(* CODESYS project CtaAppModBus_1.0.0.0.library
   Description: Modbus Library der CTA
   Version: 1.0.0.0
   Title: CtaAppModbus
   Author: SIS
   Company: CTA
   Placeholder: CtaAppModbus
   DocFormat: reStructuredText
   CompiledLibraryCompatibilityVersion: CODESYS V3.5 SP16 Patch 3
   LanguageModelAttribute: qualified-access-only
   DefaultNamespace: CtaAppModbus

Project tree, tasks and I/O mapping:
  libraries: Standard, 3.5.18.0 (System); CtaVisSymbols, 1.0.0.0 (CTA); CtaSysConfig, 1.0.0.0 (CTA); CtaAppTime, 1.0.0.0 (CTA); CtaAppBmk, 1.0.0.0 (CTA); VisuSymbols, 4.5.0.0 (System); VisuDialogs, * (System); ModbusFB, 4.3.0.0 (3S - Smart Software Solutions GmbH); IoDrvEthernet, 4.2.0.0 (3S - Smart Software Solutions GmbH); CtaVisHelp, 1.0.0.0 (CTA)
  40 Visualizations/
    HELPER/
      visualisation VIS_IP_INPUT
      visualisation VIS_IP_PARAMETER
      visualisation VIS_IP_PARAMETER_QUERRY
      visualisation VIS_IP_PARAMETER_BASE
    CLIENTMANAGER/
      LINE/
        visualisation VIS_CLIENT_LINE_QUERRY
        visualisation VIS_CLIENT_LINE
      OVERWIEV/
        visualisation VIS_CLIENT_MANAGER_OVERWIEV_QUERRY
        visualisation VIS_CLIENT_MANAGER_TABLE
        visualisation VIS_CLIENT_MANAGER_OVERWIEV
      MENÜ/
        visualisation VIS_CLIENTMANAGER_MENÜ
      visualisation DIA_CLIENT_MANAGER
      PARAMETER/
        visualisation VIS_CLIENT_MANAGER_PARAMETER
      TCP/
        PARAMETER/
          visualisation VIS_CLIENT_MANAGER_PARAMETER_TCP
          visualisation VIS_CLIENT_MANAGER_PARAMETER_TCP_QUERY
      RTU/
        PARAMETER/
          visualisation VIS_CLIENT_MANAGER_PARAMETER_RTU
          visualisation VIS_CLIENT_MANAGER_PARAMETER_RTU_QUERY
          TEXTLIST/
            text list TEXT_DTR_CONTROL
            text list TEXT_RTS_CONTROL
            text list TEXT_STOPBITS
            text list TXT_COMPORT
    MBJOB/
      visualisation VIS_JOB_QUERRY
      visualisation VIS_JOB
    CLIENT/
      TCP/
        PARAMETER/
          visualisation VIS_CLIENT_PARAMETER_TCP
          visualisation VIS_CLIENT_PARAMETER_TCP_QUERY
          visualisation VIS_CLIENT_PARAMETER_TCP_TEMP
      RTU/
        PARAMETER/
          visualisation VIS_CLIENT_PARAMETER_RTU
          visualisation VIS_CLIENT_PARAMETER_RTU_QUERY
          visualisation VIS_CLIENT_PARAMETER_RTU_TEMP
      CLIENT/
        visualisation DIA_CLIENT
        MENÜ/
          visualisation VIS_CLIENT_MENÜ
        OVERWIEV/
          visualisation VIS_CLIENT_OVERWIEV
          visualisation VIS_CLIENT_OVERWIEV_QUERY
        PARAMETER/
          visualisation VIS_CLIENT_PARAMETER
        JOBS/
          visualisation VIS_CLIENT_JOBS_TABLE
          visualisation VIS_CLIENT_JOBS_QUERRY
          visualisation VIS_CLIENT_JOBS
    SERVER/
      visualisation DIA_SERVER
  30 Program Organization Units/
    CLIENT/
      TCP/
        function block FB_MB_CLIENT_TCP [ST]: NODE_ID, ENABLE, TIMEOUT, READ_DELAY, WRITE_DELAY, IP_ADRESS, actConfig, PORT, P_fbtWriteDelay, P_fbuiPort, P_fbtTimeOut, P_fbusiNodeId, P_fbxEnable, P_fbstIpAdress, P_fbtReadDelay
      RTU/
        function block FB_MB_CLIENT_RTU [ST]: TIMEOUT, NODE_ID, READ_DELAY, WRITE_DELAY, actConfig, ENABLE, P_fbtReadDelay, P_fbtTimeOut, P_fbtWriteDelay, P_fbusiNodeId, P_fbxEnable
      BASE/
        function block FB_MB_CLIENT [ST]: ADD_MODBUS_JOB, CHECK_IF_JOB_EXIST, CREATE_JOB, GET_NEXT_JOB, DESTROY_JOB, AllJobsDone, GET_READY, BIG_SYBIL, LOW_SYBIL, SELF, CALL_AFTER_LAST_JOB_DONE, BASE_MBJOB, COUNT, ERROR, ERROR_ID, EXEPTION_CODE, AY_ITF_MBJOB_VIS, ExecuteTime, RELOAD_ARRAY, IsCurrentCall, CONFIRM_ALL_JOBS_DONE
    MBJOB/
      function block FB_MBJOB [ST]: byMbFunction, PARENT, BIG_SYBIL, pByte, wQuantity, DESTROY, wMbAdress, LOW_SYBIL, SELF
    FC/
      function FcBytePointToWordValue [ST]
      function FcBytePointToBoolValue [ST]
      function fcStringIPtoByteArray [ST]
      function fcSetInitialIPString [ST]
      function fcCheckIp [ST]
    CLIENTMANAGER/
      RTU/
        function block FB_MB_CLIENTMANAGER_RTU [ST]: actConfig, actGetError, P_fbenRTSControl, actCallFunctions, actCheckBusy, actDelays, actExecuteFunction, P_fbenStopBits, P_fbxRtuAscii, P_fbbyDataBits, P_fbdwBaudrate, P_fbenDTRControl, P_fbenParity, P_fbenPort
      TCP/
        function block FB_MB_CLIENTMANAGER_TCP [ST]: actGetError, actCheckBusy, actExecuteFunction, actDelays, actCallFunctions
      BASE/
        function block FB_MB_CLIENTMANAGER [ST]: ITF_BASE_CLIENT, ADD_MODBUS_CLIENT, CHECK_IF_EXIST, RELOAD_ARRAY, AY_ITF_MBCLIENT_VIS, OperationTime
    SERVER/
      function block fbModBusServer [ST]: actConfig, actModBusServerTcp, actModBusServerUdp, actModBusServerSerial, metGetCoil, metSetDiscretInput, metGetHoldingRegister, metSetInputRegister, metAddSerialControll, metAddTcpControll, metAddUdpControll, metSetHoldingRegister, metSetCoil
      function block FB_SERVER [ST]: actConfig, metGetCoil, metGetHoldingRegister, metSetCoil, metSetDiscretInput, metSetHoldingRegister, metSetInputRegister, actDataModel, P_Serial_fbbyDataBits, P_Serial_fbdwBaudrate, P_Serial_fbenDTRControl, P_Serial_fbenParity, P_Serial_fbenRTSControl, P_Serial_fbenStopBits, P_Serial_fbusiNodeId, P_Serial_fbxEnable, P_Serial_fbxRtuAscii, P_Serial_fbxEnableWatchDog, P_Serial_fbtWatchDog, P_Serial_fbenPort, P_Tcp_fbxEnable, P_Tcp_fbwPort, P_Tcp_fbxEnableWatchDog, P_Tcp_fbtWatchDog, P_Tcp_fbstInterface
  00000000-0000-0000-0000-000000000000|D:\CoDeSys\LibrariesV3\trunk\Intern\CAA\CAA Template\3.4.0.0 draft\Placeholder.xml
  00000000-0000-0000-0000-000000000000|D:\CoDeSys\LibrariesV3\trunk\Intern\CAA\CAA Template\3.2.0.3 draft\Prefix.pdf
  00000000-0000-0000-0000-000000000000|D:\CoDeSys\LibrariesV3\trunk\Intern\CAA\CAA Template\3.5.2.0 draft\Placeholder.xml
  20 Structs/
    SERVER/
      PARAMETER/
        data type scModBusServerParameter
        TCP/
          data type scTcp
        SERIAL/
          data type scSerial
    CLIENT/
      NETWORK/
        data type scTcpClientParameter
      SERIAL/
        data type scSerialPortParameter
        data type scSerialClientParameter
  50 Images/
  10 Documenation/
    global variables VersionHistory
    global variables readMe
  21 Interface/
    CLIENTMANAGER/
      RTU/
        interface ITF_MB_CLIENTMANAGER_RTU: P_fbenStopBits, P_fbenPort, P_fbdwBaudrate, P_fbbyDataBits, P_fbenParity, P_fbenDTRControl, P_fbenRTSControl, P_fbxRtuAscii
      BASE/
        interface ITF_MB_CLIENTMANAGER: OperationTime, ITF_BASE_CLIENT, AY_ITF_MBCLIENT_VIS, RELOAD_ARRAY
      TCP/
        interface ITF_MB_CLIENTMANAGER_TCP
    MBJOB/
      interface ITF_MBJOB: PARENT, DESTROY, BIG_SYBIL, LOW_SYBIL, SELF, byMbFunction, pByte, wMbAdress, wQuantity
    CLIENT/
      BASE/
        interface ITF_CLIENT: CHECK_IF_JOB_EXIST, CREATE_JOB, DESTROY_JOB, GET_NEXT_JOB, GET_READY, AllJobsDone, BIG_SYBIL, LOW_SYBIL, SELF, BASE_MBJOB, COUNT, ADD_MODBUS_JOB, ERROR, ERROR_ID, EXEPTION_CODE, AY_ITF_MBJOB_VIS, ExecuteTime, RELOAD_ARRAY, IsCurrentCall, CONFIRM_ALL_JOBS_DONE, CALL_AFTER_LAST_JOB_DONE
      RTU/
        interface ITF_MB_CLIENT_RTU: ENABLE, P_fbxEnable, P_fbusiNodeId, P_fbtTimeOut, P_fbtReadDelay, P_fbtWriteDelay, NODE_ID, TIMEOUT, READ_DELAY, WRITE_DELAY
      TCP/
        interface ITF_MB_CLIENT_TCP: ENABLE, NODE_ID, TIMEOUT, READ_DELAY, WRITE_DELAY, IP_ADRESS, PORT, P_fbxEnable, P_fbusiNodeId, P_fbtTimeOut, P_fbtReadDelay, P_fbtWriteDelay, P_fbuiPort, P_fbstIpAdress
    SERVER/
      interface ITF_SERVER: metGetCoil, metGetHoldingRegister, metSetCoil, metSetDiscretInput, metSetHoldingRegister, metSetInputRegister
      interface ITF_SERVER_PARA: P_Serial_fbxEnable, P_Serial_fbusiNodeId, P_Serial_fbdwBaudrate, P_Serial_fbbyDataBits, P_Serial_fbenParity, P_Serial_fbenStopBits, P_Serial_fbenDTRControl, P_Serial_fbenRTSControl, P_Serial_fbxRtuAscii, P_Serial_fbxEnableWatchDog, P_Serial_fbtWatchDog, P_Serial_fbenPort, P_Tcp_fbxEnable, P_Tcp_fbwPort, P_Tcp_fbxEnableWatchDog, P_Tcp_fbtWatchDog, P_Tcp_fbstInterface
  11 Library Parameter/
  12 Konstanten/
  60 Textlisten/
    SERIAL/
      text list txtPhysikalLayer
      text list txtParity
      text list txtHandshake
      text list txtStopBits
  13 Globale Variablen/
  text list GlobalTextList
*)

// 20 Structs/SERVER/PARAMETER/scModBusServerParameter
TYPE scModBusServerParameter :
    STRUCT
        scSerial    :   scSerial;
        scTcp       :   scTcp;
    END_STRUCT
END_TYPE

// 20 Structs/SERVER/PARAMETER/TCP/scTcp
TYPE scTcp :
    STRUCT
        fbxEnable           :   CtaSysConfig.fbBOOL;           // Tcp Server Enable    
        fbwPort             :   CtaSysConfig.fbWORD;           // Tcp Server Port
        fbxEnableWatchDog   :   CtaSysConfig.fbBOOL;           // WatchDog Enable
        fbtWatchDog         :   CtaSysConfig.fbTIME;           // WatchDog Time
		fbstInterface		:	CtaSysConfig.fbSTRING40;	   // Interface Name
    END_STRUCT
END_TYPE

// 20 Structs/SERVER/PARAMETER/SERIAL/scSerial
TYPE scSerial :
    STRUCT
        fbxEnable           				:   CtaSysConfig.fbBOOL;        // Serial Server Enable
        fbxEnableWatchDog   				:   CtaSysConfig.fbBOOL;        // WatchDog Enable
        fbtWatchDog         				:   CtaSysConfig.fbTIME;        // WatchDog Time		
		fbenPort							:	CtaSysConfig.fbINT;			// PORT NONE , COM1, COM2 ...
		fbusiNodeId							:	CtaSysConfig.fbUSINT;      	// Serial Server Id  
		fbdwBaudrate						:	CtaSysConfig.fbDWORD;		// Baudrate 
		fbbyDataBits						:	CtaSysConfig.fbBYTE;		// Data Bits
		fbenParity							:	CtaSysConfig.fbBYTE;		// Parity
		fbenStopBits						:	CtaSysConfig.fbBYTE;		// Stopbits
		fbenDTRControl						:	CtaSysConfig.fbBYTE;		// DTR Control
		fbenRTSControl						:	CtaSysConfig.fbBYTE;		// RTS Control
		fbxRtuAscii							:	CtaSysConfig.fbBOOL;		// RTU = FALSE , ASCII = TRUE
    END_STRUCT
END_TYPE

// 20 Structs/CLIENT/NETWORK/scTcpClientParameter
TYPE scTcpClientParameter :
    STRUCT
        fbxEnable					:	CtaSysConfig.fbBOOL;        // Serial Server Enable       
        fbusiNodeId					:	CtaSysConfig.fbUSINT;     	// Serial Server Id  
        fbtTimeOut					:	CtaSysConfig.fbTIME;        // Timeout Time
        fbtReadDelay				:	CtaSysConfig.fbTIME;      	// Read Delay        
        fbtWriteDelay				:	CtaSysConfig.fbTIME;     	// Write Delay 	
		fbuiPort					:	CtaSysConfig.fbUINT;      	// Port Nr  
		fbstIpAdress				:	CtaSysConfig.fbSTRING40;    // IP Adresse   
    END_STRUCT
END_TYPE

// 20 Structs/CLIENT/SERIAL/scSerialPortParameter
TYPE scSerialPortParameter :
    STRUCT 
		fbenPort							:	CtaSysConfig.fbINT;			// PORT NONE , COM1, COM2 ...
		fbdwBaudrate						:	CtaSysConfig.fbDWORD;		// Baudrate 
		fbbyDataBits						:	CtaSysConfig.fbBYTE;		// Data Bits
		fbenParity							:	CtaSysConfig.fbBYTE;		// Parity
		fbenStopBits						:	CtaSysConfig.fbBYTE;		// Stopbits
		fbenDTRControl						:	CtaSysConfig.fbBYTE;		// DTR Control
		fbenRTSControl						:	CtaSysConfig.fbBYTE;		// RTS Control
		fbxRtuAscii							:	CtaSysConfig.fbBOOL;		// RTU = FALSE , ASCII = TRUE
    END_STRUCT
END_TYPE

// 20 Structs/CLIENT/SERIAL/scSerialClientParameter
TYPE scSerialClientParameter :
    STRUCT
        fbxEnable					:	CtaSysConfig.fbBOOL;       // Serial Server Enable        
        fbusiNodeId					:	CtaSysConfig.fbUSINT;      // Serial Server Id        
        fbtTimeOut					:	CtaSysConfig.fbTIME;       // Timeout Time
		fbtReadDelay				:	CtaSysConfig.fbTIME; 	   // Read Delay
		fbtWriteDelay				:	CtaSysConfig.fbTIME;	   // Write Delay
    END_STRUCT
END_TYPE

// 10 Documenation/VersionHistory
(* 

.. image:: ../../Images/CTA_Logo.jpg
   :align: right
   :width: 15% 

**Vorlage**   


============ =========== =========== ============================================
**Date**     **Version** **Author**  **Change**
------------ ----------- ----------- --------------------------------------------
04.03.2021   0.0.0.0     SIS         Vorlage erstellt

============ =========== =========== ============================================


*)
VAR_GLOBAL
    stInfo : STRING:= '0.0.0.0, Vorlage, CTA';
END_VAR

// 10 Documenation/readMe
(*

**ReadMe**
 
|	**Empfehlung**
|
|	Dokumentrieren Sie die Library für eine nachhaltige Entwicklung
|     
| *Beispiel* 
|
| Dies ist die Vorlage Library der CTA. Erstellen Sie ihre Library anhand dieser Vorlage.
*)

VAR_GLOBAL
    xReadMeDone              :   BOOL;
END_VAR

// 30 Program Organization Units/MBJOB/FB_MBJOB
{attribute 'enable_dynamic_creation'}
FUNCTION_BLOCK FB_MBJOB IMPLEMENTS ITF_MBJOB
VAR_OUTPUT
END_VAR
VAR
	_xConfirmExecute:	BOOL;
	_byMbFunction	:	BYTE;
	_wMbAdress		:	WORD;
	_pByte			:	POINTER TO BYTE;
	_wQuantity		:	WORD;	
	_ITF_BIG_SYBIL	:	ITF_MBJOB;
	_ITF_LOW_SYBIL	:	ITF_MBJOB;
	_ITF_PARENT		:	ITF_CLIENT;
END_VAR

PROPERTY byMbFunction : BYTE
GET
byMbFunction := _byMbFunction;
END_GET
SET
_byMbFunction := byMbFunction;
END_SET
END_PROPERTY

PROPERTY PARENT : ITF_CLIENT
SET
_ITF_PARENT := PARENT;
END_SET
END_PROPERTY

{attribute 'estimated-stack-usage' := '104'}
PROPERTY BIG_SYBIL : ITF_MBJOB
GET
BIG_SYBIL := _ITF_BIG_SYBIL;
END_GET
SET
_ITF_BIG_SYBIL := BIG_SYBIL;
IF __QUERYINTERFACE(_ITF_BIG_SYBIL,_ITF_BIG_SYBIL) THEN
	IF _ITF_BIG_SYBIL.LOW_SYBIL <> SELF THEN
		_ITF_BIG_SYBIL.LOW_SYBIL := THIS^;
	END_IF;
END_IF;
END_SET
END_PROPERTY

PROPERTY pByte : POINTER TO BYTE
GET
pByte := _pByte;
END_GET
SET
_pByte := pByte;
END_SET
END_PROPERTY

PROPERTY wQuantity : WORD
GET
wQuantity := _wQuantity;
END_GET
SET
_wQuantity := wQuantity;
END_SET
END_PROPERTY

METHOD DESTROY
VAR
	pSelf	:	POINTER TO FB_MBJOB;
END_VAR
IF __QUERYINTERFACE(_ITF_BIG_SYBIL,_ITF_BIG_SYBIL) THEN
	_ITF_BIG_SYBIL.LOW_SYBIL := _ITF_LOW_SYBIL;
END_IF;

IF __QUERYINTERFACE(_ITF_LOW_SYBIL,_ITF_LOW_SYBIL) THEN
	_ITF_LOW_SYBIL.BIG_SYBIL := _ITF_BIG_SYBIL;
END_IF;

IF __QUERYINTERFACE(_ITF_PARENT,_ITF_PARENT) THEN
	_ITF_PARENT.RELOAD_ARRAY(TRUE,FALSE,FALSE);
END_IF;

pSelf := THIS;

__DELETE(pSelf);
END_METHOD

PROPERTY wMbAdress : WORD
SET
_wMbAdress := wMbAdress;
END_SET
GET
wMbAdress := _wMbAdress;
END_GET
END_PROPERTY

{attribute 'estimated-stack-usage' := '104'}
PROPERTY LOW_SYBIL : ITF_MBJOB
GET
LOW_SYBIL := _ITF_LOW_SYBIL;
END_GET
SET
_ITF_LOW_SYBIL := LOW_SYBIL;
IF __QUERYINTERFACE(_ITF_LOW_SYBIL,_ITF_LOW_SYBIL) THEN
	IF _ITF_LOW_SYBIL.BIG_SYBIL <> SELF THEN
		_ITF_LOW_SYBIL.BIG_SYBIL := THIS^;
	END_IF;
END_IF;
END_SET
END_PROPERTY

PROPERTY SELF : ITF_MBJOB
GET
SELF := THIS^;
END_GET
END_PROPERTY

END_FUNCTION_BLOCK

// 21 Interface/MBJOB/ITF_MBJOB
INTERFACE ITF_MBJOB EXTENDS __System.IQUERYINTERFACE

PROPERTY PARENT : ITF_CLIENT
SET
END_SET
END_PROPERTY

METHOD DESTROY
END_METHOD

PROPERTY BIG_SYBIL : ITF_MBJOB
GET
END_GET
SET
END_SET
END_PROPERTY

PROPERTY LOW_SYBIL : ITF_MBJOB
GET
END_GET
SET
END_SET
END_PROPERTY

PROPERTY SELF : ITF_MBJOB
GET
END_GET
END_PROPERTY

PROPERTY byMbFunction : BYTE
SET
END_SET
GET
END_GET
END_PROPERTY

PROPERTY pByte : POINTER TO BYTE
SET
END_SET
GET
END_GET
END_PROPERTY

PROPERTY wMbAdress : WORD
SET
END_SET
GET
END_GET
END_PROPERTY

PROPERTY wQuantity : WORD
GET
END_GET
SET
END_SET
END_PROPERTY

END_INTERFACE

// 21 Interface/CLIENT/BASE/ITF_CLIENT
INTERFACE ITF_CLIENT  EXTENDS CtaAppBmk.ITF_BMK

METHOD CHECK_IF_JOB_EXIST : BOOL
VAR_INPUT
	_byMbFunction	:	BYTE;
	_wMbAdress		:	WORD;
	_pByte			:	POINTER TO BYTE;
	_wQuantity		:	WORD;	
END_VAR
END_METHOD

METHOD CREATE_JOB : BOOL
VAR_INPUT
	_byMbFunction	:	BYTE;
	_wMbAdress		:	WORD;
	_pData			:	POINTER TO BYTE;
	_wQuantity		:	WORD;		
END_VAR
END_METHOD

METHOD DESTROY_JOB : BOOL
VAR_INPUT
	_byMbFunction	:	BYTE;
	_wMbAdress		:	WORD;
	_pData			:	POINTER TO BYTE;
	_wQuantity		:	WORD;		
END_VAR
END_METHOD

METHOD GET_NEXT_JOB : BOOL
VAR_OUTPUT
	_byMbFunction	:	BYTE;
	_wMbAdress		:	WORD;
	_pByte			:	POINTER TO BYTE;
	_wQuantity		:	WORD;	
END_VAR
END_METHOD

METHOD GET_READY : BOOL
VAR_INPUT
END_VAR
END_METHOD

PROPERTY AllJobsDone : BOOL
GET
END_GET
END_PROPERTY

PROPERTY BIG_SYBIL : ITF_CLIENT
GET
END_GET
SET
END_SET
END_PROPERTY

PROPERTY LOW_SYBIL : ITF_CLIENT
GET
END_GET
SET
END_SET
END_PROPERTY

PROPERTY SELF : ITF_CLIENT
GET
END_GET
END_PROPERTY

PROPERTY BASE_MBJOB : ITF_MBJOB
GET
END_GET
END_PROPERTY

PROPERTY COUNT : UINT
GET
END_GET
END_PROPERTY

METHOD ADD_MODBUS_JOB
VAR_INPUT
	ITF_MBJOB_IN	:	ITF_MBJOB;
END_VAR
END_METHOD

PROPERTY ERROR : BOOL
SET
END_SET
GET
END_GET
END_PROPERTY

PROPERTY ERROR_ID : ModbusFB.Error
SET
END_SET
GET
END_GET
END_PROPERTY

PROPERTY EXEPTION_CODE : ModbusFB.ExceptionCodes
SET
END_SET
GET
END_GET
END_PROPERTY

PROPERTY AY_ITF_MBJOB_VIS : ARRAY[0..9] OF ITF_MBJOB
GET
END_GET
END_PROPERTY

PROPERTY ExecuteTime : LTIME
GET
END_GET
END_PROPERTY

METHOD RELOAD_ARRAY
VAR_INPUT
	xInit				:	BOOL;
	xLoadNext10			:	BOOL;
	xLoadLast10			:	BOOL;
END_VAR
END_METHOD

PROPERTY IsCurrentCall : BOOL
GET
END_GET
END_PROPERTY

PROPERTY CONFIRM_ALL_JOBS_DONE : BOOL
GET
END_GET
END_PROPERTY

METHOD CALL_AFTER_LAST_JOB_DONE
VAR_INPUT
END_VAR
END_METHOD

END_INTERFACE

// 30 Program Organization Units/CLIENT/TCP/FB_MB_CLIENT_TCP
FUNCTION_BLOCK FB_MB_CLIENT_TCP EXTENDS FB_MB_CLIENT IMPLEMENTS ITF_MB_CLIENT_TCP
VAR_OUTPUT
END_VAR
VAR
	(* Config *)
	fbConfigFile				:	CtaSysConfig.fbConfigFile;
	scParameter                	: 	scTcpClientParameter;
END_VAR

(* Config File *)
actConfig();

PROPERTY NODE_ID : USINT
GET
NODE_ID := scParameter.fbusiNodeId.proValue;
END_GET
END_PROPERTY

PROPERTY ENABLE : BOOL
GET
ENABLE := scParameter.fbxEnable.proValue;
END_GET
END_PROPERTY

PROPERTY TIMEOUT : TIME
GET
TIMEOUT := scParameter.fbtTimeOut.proValue;
END_GET
END_PROPERTY

PROPERTY READ_DELAY : TIME
GET
READ_DELAY := scParameter.fbtReadDelay.proValue;
END_GET
END_PROPERTY

PROPERTY WRITE_DELAY : TIME
GET
WRITE_DELAY := scParameter.fbtWriteDelay.proValue;
END_GET
END_PROPERTY

PROPERTY IP_ADRESS : STRING(15)
GET
IP_ADRESS := scParameter.fbstIpAdress.proValue;
END_GET
END_PROPERTY

ACTION actConfig:
(* Config File *)
fbConfigFile();

scParameter.fbxEnable		(_usiParaNr := 1,itfConfigFb := fbConfigFile										);		
scParameter.fbusiNodeId		(_usiParaNr := 2,itfConfigFb := fbConfigFile,_MinInit := 0	  , _MaxInit := 255		);		
scParameter.fbtTimeOut		(_usiParaNr := 3,itfConfigFb := fbConfigFile,_MinInit := T#0MS, _MaxInit := T#5M 	);		
scParameter.fbtReadDelay	(_usiParaNr := 4,itfConfigFb := fbConfigFile,_MinInit := T#0MS, _MaxInit := T#5M 	);		
scParameter.fbtWriteDelay	(_usiParaNr := 5,itfConfigFb := fbConfigFile,_MinInit := T#0MS, _MaxInit := T#5M 	);	
scParameter.fbuiPort		(_usiParaNr := 6,itfConfigFb := fbConfigFile										);
scParameter.fbstIpAdress	(_usiParaNr := 7,itfConfigFb := fbConfigFile										);

(* Check Ip *)
IF scParameter.fbstIpAdress.proStateChanged THEN
	IF NOT fcCheckIp(scParameter.fbstIPAdress.proValue) THEN
		fcSetInitialIPString(scParameter.fbstIpAdress);
	END_IF;
END_IF;
END_ACTION

PROPERTY PORT : UINT
GET
PORT := scParameter.fbuiPort.proValue;
END_GET
END_PROPERTY

PROPERTY P_fbtWriteDelay : CtaSysConfig.ITF_DATATYPE
GET
P_fbtWriteDelay := scParameter.fbtWriteDelay;
END_GET
END_PROPERTY

PROPERTY P_fbuiPort : CtaSysConfig.ITF_DATATYPE
GET
P_fbuiPort := scParameter.fbuiPort;
END_GET
END_PROPERTY

PROPERTY P_fbtTimeOut : CtaSysConfig.ITF_DATATYPE
GET
P_fbtTimeOut := scParameter.fbtTimeOut;
END_GET
END_PROPERTY

PROPERTY P_fbusiNodeId : CtaSysConfig.ITF_DATATYPE
GET
P_fbusiNodeId := scParameter.fbusiNodeId;
END_GET
END_PROPERTY

PROPERTY P_fbxEnable : CtaSysConfig.ITF_DATATYPE
GET
P_fbxEnable := scParameter.fbxEnable;
END_GET
END_PROPERTY

PROPERTY P_fbstIpAdress : CtaSysConfig.ITF_DATATYPE
GET
P_fbstIpAdress := scParameter.fbstIpAdress;
END_GET
END_PROPERTY

PROPERTY P_fbtReadDelay : CtaSysConfig.ITF_DATATYPE
GET
P_fbtReadDelay := scParameter.fbtReadDelay;
END_GET
END_PROPERTY

END_FUNCTION_BLOCK

// 30 Program Organization Units/CLIENT/BASE/FB_MB_CLIENT
FUNCTION_BLOCK FB_MB_CLIENT EXTENDS CtaAppBmk.fbBMK IMPLEMENTS ITF_CLIENT
VAR_OUTPUT
	udiDynMem					:	UDINT;
	xAllJobsDone				:	BOOL;
	xConfirmAllJobsDone			:	BOOL;
END_VAR             			
VAR                 			
	_ITF_BIG_SYBIL				:	ITF_CLIENT;
	_ITF_LOW_SYBIL				:	ITF_CLIENT;
	                			
	_BASE_MBU_JOB				:	ITF_MBJOB;
	_TEMP_REG_JOB				:	ITF_MBJOB;
	_TEMP_MBU_JOB				:	ITF_MBJOB;	
	
	_COUNT						:	UINT;
	_udiDynMemTemp				:	UDINT;
	xGetReadyCalled				:	BOOL;
	xNoChangeHappen				:	BOOL;
	
	xErrorHappen				:	BOOL;
	eErrorID					:	ModbusFB.Error;
	eExeptionCode				:	ModbusFB.ExceptionCodes;
	
	fbTimeStop					:	CtaAppTime.fbTimeMeasurement;
	ltTime						:	LTIME;
	
	_ayITF_MBJOB_VIS			:	ARRAY[0..9] OF ITF_MBJOB;
END_VAR

METHOD ADD_MODBUS_JOB
VAR_INPUT
	ITF_MBJOB_IN	:	ITF_MBJOB;
END_VAR
VAR
	ITF_TEMP		:	ITF_MBJOB;
	ITF_TEMP_BIG	:	ITF_MBJOB;
	ITF_TEMP_LOW	:	ITF_MBJOB;
	xDone			:	BOOL;
END_VAR
(* Check if Valid Interface Input *)
IF __QUERYINTERFACE(ITF_MBJOB_IN,ITF_MBJOB_IN) THEN
	ITF_MBJOB_IN.PARENT := THIS^;
	(* Check if Valid Interface Base*)
	IF __QUERYINTERFACE(_BASE_MBU_JOB,_BASE_MBU_JOB) THEN
		(* Check if Valid Interface Temporary registration *)
		IF __QUERYINTERFACE(_TEMP_REG_JOB,ITF_TEMP) THEN
			REPEAT
				(* Get Big Sybil of registration *)
				IF __QUERYINTERFACE(ITF_TEMP.BIG_SYBIL,ITF_TEMP_BIG) THEN
					(* Check if Function Code is Lower or Bigger *)
					IF ITF_MBJOB_IN.byMbFunction <= ITF_TEMP.byMbFunction AND
						ITF_MBJOB_IN.byMbFunction >= ITF_TEMP_BIG.byMbFunction THEN
						(* Check if Adress is Lower *)
						IF ITF_MBJOB_IN.wMbAdress <= ITF_TEMP.wMbAdress THEN
							(* Check if Adress is Bigger and update if yes*)
							IF ITF_MBJOB_IN.wMbAdress >= ITF_TEMP_BIG.wMbAdress THEN
								ITF_MBJOB_IN.BIG_SYBIL := ITF_TEMP.BIG_SYBIL;
								ITF_MBJOB_IN.LOW_SYBIL := ITF_TEMP;
								xDone	 := TRUE;							
							END_IF;
						(* Adress is Bigger update *)
						ELSE
							IF __QUERYINTERFACE(ITF_TEMP.LOW_SYBIL,ITF_TEMP_LOW) THEN
								IF ITF_MBJOB_IN.byMbFunction < ITF_TEMP_LOW.byMbFunction OR
									(ITF_MBJOB_IN.byMbFunction = ITF_TEMP_LOW.byMbFunction AND
									ITF_MBJOB_IN.wMbAdress <= ITF_TEMP_LOW.wMbAdress) THEN
									ITF_MBJOB_IN.LOW_SYBIL := ITF_TEMP.LOW_SYBIL;
									ITF_MBJOB_IN.BIG_SYBIL := ITF_TEMP;
									xDone	 := TRUE;
								END_IF;
							ELSE
								ITF_MBJOB_IN.LOW_SYBIL := ITF_TEMP.LOW_SYBIL;
								ITF_MBJOB_IN.BIG_SYBIL := ITF_TEMP;
								xDone	 := TRUE;
								(* Update Registation Job if temp is the last one *)
								IF ITF_TEMP = _TEMP_REG_JOB THEN
									_TEMP_REG_JOB := ITF_MBJOB_IN;
									_TEMP_REG_JOB.LOW_SYBIL := 0;
								END_IF;
							END_IF;
						END_IF;
					(* Function Code ist Bigger Insert after temporary*)
					ELSIF ITF_MBJOB_IN.byMbFunction > ITF_TEMP.byMbFunction THEN
						ITF_MBJOB_IN.LOW_SYBIL := ITF_TEMP.LOW_SYBIL;
						ITF_MBJOB_IN.BIG_SYBIL := ITF_TEMP;
						xDone	 := TRUE;
						(* Update Registation Job if temp is the last one *)
						IF ITF_TEMP = _TEMP_REG_JOB THEN
							_TEMP_REG_JOB := ITF_MBJOB_IN;
							_TEMP_REG_JOB.LOW_SYBIL := 0;
						END_IF
					END_IF;
				(* Interface is same as the Base*)
				ELSIF ITF_TEMP = _BASE_MBU_JOB THEN
					(* Check if the Input Interface needs to be the new base*)
					IF ITF_MBJOB_IN.byMbFunction <= ITF_TEMP.byMbFunction AND
						ITF_MBJOB_IN.wMbAdress <= ITF_TEMP.wMbAdress THEN 
						ITF_MBJOB_IN.LOW_SYBIL := ITF_TEMP;
						_BASE_MBU_JOB := ITF_MBJOB_IN;
						_BASE_MBU_JOB.BIG_SYBIL := 0;
						xDone	 := TRUE; 
					ELSE
						(* Update Registation Job if temp is the last one *)
						IF ITF_TEMP = _TEMP_REG_JOB THEN
							_TEMP_REG_JOB := ITF_MBJOB_IN;
							_TEMP_REG_JOB.LOW_SYBIL := 0;
						END_IF
						ITF_MBJOB_IN.LOW_SYBIL := _BASE_MBU_JOB.LOW_SYBIL;
						_BASE_MBU_JOB.LOW_SYBIL := ITF_MBJOB_IN;
					END_IF;
				END_IF;
				(* Get Next Interface to Check*)
				__QUERYINTERFACE(ITF_TEMP.BIG_SYBIL,ITF_TEMP);
			UNTIL xDone OR ITF_TEMP = 0 
			END_REPEAT
		ELSE
			(* Set Base Low sybill on second call*)
			_BASE_MBU_JOB.LOW_SYBIL := ITF_MBJOB_IN;
			_TEMP_REG_JOB := ITF_MBJOB_IN;		
		END_IF;		
	ELSE
		(* Set Base on first call*)
		_BASE_MBU_JOB := ITF_MBJOB_IN;
		_TEMP_REG_JOB := ITF_MBJOB_IN;
	END_IF;
	(* Count Jobs *)
	_COUNT := _COUNT + 1;
	THIS^.RELOAD_ARRAY(TRUE,FALSE,FALSE);
END_IF;
END_METHOD

METHOD CHECK_IF_JOB_EXIST : BOOL
VAR_INPUT
	_byMbFunction	:	BYTE;
	_wMbAdress		:	WORD;
	_pByte			:	POINTER TO BYTE;
	_wQuantity		:	WORD;	
END_VAR
VAR
	_TEMP_CHK_JOB	:	ITF_MBJOB;
	udiSafe			:	UDINT;
END_VAR
IF __QUERYINTERFACE(_BASE_MBU_JOB,_TEMP_CHK_JOB) THEN
	REPEAT 
		IF _TEMP_CHK_JOB.byMbFunction = _byMbFunction AND
			_TEMP_CHK_JOB.wMbAdress	= _wMbAdress AND
			_TEMP_CHK_JOB.pByte = _pByte AND
			_TEMP_CHK_JOB.wQuantity = _wQuantity THEN
			CHECK_IF_JOB_EXIST := TRUE;
		END_IF;
		_TEMP_CHK_JOB := _TEMP_CHK_JOB.LOW_SYBIL;
		udiSafe	:= udiSafe + 1;
	UNTIL CHECK_IF_JOB_EXIST OR _TEMP_CHK_JOB = 0 OR udiSafe >= 16#FFFFFFFE
	END_REPEAT
ELSE
	CHECK_IF_JOB_EXIST := FALSE;
END_IF
END_METHOD

METHOD CREATE_JOB : BOOL
VAR_INPUT
	_byMbFunction	:	BYTE;
	_wMbAdress		:	WORD;
	_pData			:	POINTER TO BYTE;
	_wQuantity		:	WORD;		
END_VAR
VAR	
	pFbMbJob		:	POINTER TO FB_MBJOB;
END_VAR
IF _pData <> 0 THEN
	IF NOT CHECK_IF_JOB_EXIST(_byMbFunction,_wMbAdress,_pData,_wQuantity) THEN
		pFbMbJob := __NEW(FB_MBJOB);
		IF pFbMbJob <> 0 THEN
			_udiDynMemTemp 			:= _udiDynMemTemp + SIZEOF(FB_MBJOB);
			udiDynMem				:= MAX(udiDynMem,_udiDynMemTemp);
			pFbMbJob^.byMbFunction 	:= _byMbFunction;
			pFbMbJob^.wMbAdress	 	:= _wMbAdress;
			pFbMbJob^.pByte		 	:= _pData;
			pFbMbJob^.wQuantity 	:= _wQuantity;
			ADD_MODBUS_JOB(pFbMbJob^);
			xNoChangeHappen			:= FALSE;
			xConfirmAllJobsDone		:= FALSE;
		END_IF;
	END_IF;
END_IF;
END_METHOD

METHOD GET_NEXT_JOB : BOOL
VAR_OUTPUT
	_byMbFunction	:	BYTE;
	_wMbAdress		:	WORD;
	_pByte			:	POINTER TO BYTE;
	_wQuantity		:	WORD;	
END_VAR
IF xGetReadyCalled THEN 
	IF __QUERYINTERFACE(_TEMP_MBU_JOB,_TEMP_MBU_JOB) THEN
		_byMbFunction		:= _TEMP_MBU_JOB.byMbFunction;
		_wMbAdress			:= _TEMP_MBU_JOB.wMbAdress;
		_pByte				:= _TEMP_MBU_JOB.pByte;
		_wQuantity			:= _TEMP_MBU_JOB.wQuantity;	
		_TEMP_MBU_JOB		:= _TEMP_MBU_JOB.LOW_SYBIL;
		GET_NEXT_JOB		:= TRUE;
		IF NOT __QUERYINTERFACE(_TEMP_MBU_JOB,_TEMP_MBU_JOB) THEN
			xAllJobsDone 	:= TRUE;
			xGetReadyCalled := FALSE;
			ltTime			:= fbTimeStop.Stop();
		END_IF;
	ELSIF  __QUERYINTERFACE(_BASE_MBU_JOB,_TEMP_MBU_JOB) THEN 	
		_byMbFunction		:= _TEMP_MBU_JOB.byMbFunction;
		_wMbAdress			:= _TEMP_MBU_JOB.wMbAdress;
		_pByte				:= _TEMP_MBU_JOB.pByte;
		_wQuantity			:= _TEMP_MBU_JOB.wQuantity;
		GET_NEXT_JOB    	:= TRUE;
		fbTimeStop.Start();
	END_IF;
END_IF;
END_METHOD

METHOD DESTROY_JOB : BOOL
VAR_INPUT
	_byMbFunction	:	BYTE;
	_wMbAdress		:	WORD;
	_pData			:	POINTER TO BYTE;
	_wQuantity		:	WORD;		
END_VAR
VAR	
	udiSafe			:	UDINT;
	_TEMP_DES_JOB	:	ITF_MBJOB;
END_VAR
IF __QUERYINTERFACE(_BASE_MBU_JOB,_TEMP_DES_JOB) THEN
	REPEAT 
		IF _TEMP_DES_JOB.byMbFunction = _byMbFunction AND
			_TEMP_DES_JOB.wMbAdress	= _wMbAdress AND
			_TEMP_DES_JOB.pByte = _pData AND
			_TEMP_DES_JOB.wQuantity = _wQuantity THEN
			IF _TEMP_DES_JOB = _TEMP_REG_JOB THEN
				_TEMP_REG_JOB := _TEMP_DES_JOB.BIG_SYBIL;
			END_IF;
			IF _TEMP_DES_JOB = _BASE_MBU_JOB THEN
				_BASE_MBU_JOB := _TEMP_DES_JOB.LOW_SYBIL;
				IF NOT __QUERYINTERFACE(_BASE_MBU_JOB,_BASE_MBU_JOB) THEN
					_TEMP_REG_JOB := _BASE_MBU_JOB;
				END_IF;
			END_IF;
			_TEMP_DES_JOB.DESTROY();
			_COUNT 			:= _COUNT -1;
			_udiDynMemTemp 	:= _udiDynMemTemp - SIZEOF(FB_MBJOB);
			DESTROY_JOB 	:= TRUE;
		ELSE
			_TEMP_DES_JOB := _TEMP_DES_JOB.LOW_SYBIL;
		END_IF;
		udiSafe	:= udiSafe + 1;
	UNTIL DESTROY_JOB OR _TEMP_DES_JOB = 0 OR udiSafe >= 16#FFFFFFFE
	END_REPEAT
ELSE
	DESTROY_JOB := FALSE;
END_IF
END_METHOD

PROPERTY AllJobsDone : BOOL
GET
AllJobsDone := xAllJobsDone;
END_GET
END_PROPERTY

METHOD GET_READY : BOOL
VAR_INPUT
END_VAR
xGetReadyCalled := TRUE;
xNoChangeHappen := TRUE;
xAllJobsDone	:= FALSE;
_TEMP_MBU_JOB   := 0;
END_METHOD

{attribute 'estimated-stack-usage' := '104'}
PROPERTY BIG_SYBIL : ITF_CLIENT
GET
BIG_SYBIL := _ITF_BIG_SYBIL;
END_GET
SET
_ITF_BIG_SYBIL := BIG_SYBIL;
IF __QUERYINTERFACE(_ITF_BIG_SYBIL,_ITF_BIG_SYBIL) THEN
	IF _ITF_BIG_SYBIL.LOW_SYBIL <> SELF THEN
		_ITF_BIG_SYBIL.LOW_SYBIL := THIS^;
	END_IF;
END_IF;
END_SET
END_PROPERTY

{attribute 'estimated-stack-usage' := '104'}
PROPERTY LOW_SYBIL : ITF_CLIENT
GET
LOW_SYBIL := _ITF_LOW_SYBIL;
END_GET
SET
_ITF_LOW_SYBIL := LOW_SYBIL;
IF __QUERYINTERFACE(_ITF_LOW_SYBIL,_ITF_LOW_SYBIL) THEN
	IF _ITF_LOW_SYBIL.BIG_SYBIL <> SELF THEN
		_ITF_LOW_SYBIL.BIG_SYBIL := THIS^;
	END_IF;
END_IF;
END_SET
END_PROPERTY

PROPERTY SELF : ITF_CLIENT
GET
SELF := THIS^;
END_GET
END_PROPERTY

METHOD CALL_AFTER_LAST_JOB_DONE
VAR_INPUT
END_VAR
xConfirmAllJobsDone := xNoChangeHappen;
END_METHOD

PROPERTY BASE_MBJOB : ITF_MBJOB
GET
BASE_MBJOB := _BASE_MBU_JOB;
END_GET
END_PROPERTY

PROPERTY COUNT : UINT
GET
COUNT := _COUNT;
END_GET
END_PROPERTY

PROPERTY ERROR : BOOL
GET
ERROR := xErrorHappen;
END_GET
SET
xErrorHappen := ERROR;
END_SET
END_PROPERTY

PROPERTY ERROR_ID : ModbusFB.Error
SET
eErrorID := ERROR_ID;
END_SET
GET
ERROR_ID := eErrorID;
END_GET
END_PROPERTY

PROPERTY EXEPTION_CODE : ModbusFB.ExceptionCodes
SET
eExeptionCode := EXEPTION_CODE;
END_SET
GET
EXEPTION_CODE := eExeptionCode;
END_GET
END_PROPERTY

PROPERTY AY_ITF_MBJOB_VIS : ARRAY[0..9] OF ITF_MBJOB
GET
AY_ITF_MBJOB_VIS := _ayITF_MBJOB_VIS;
END_GET
END_PROPERTY

PROPERTY ExecuteTime : LTIME
GET
ExecuteTime := ltTime;
END_GET
END_PROPERTY

METHOD RELOAD_ARRAY
VAR_INPUT
	xInit				:	BOOL;
	xLoadNext10			:	BOOL;
	xLoadLast10			:	BOOL;
END_VAR
VAR
	diFor				:	DINT;
	ITF_TEMP_MBJOB_VIS	:	ITF_MBJOB;
	ITF_TEMP_SAFE		:	ITF_MBJOB;
	ITF_TEMP_LAST_VALID	:	ITF_MBJOB;
END_VAR
(* Init Array *)
IF xInit THEN
	_ayITF_MBJOB_VIS[LOWER_BOUND(_ayITF_MBJOB_VIS,1)] := _BASE_MBU_JOB;
	FOR diFor := LOWER_BOUND(_ayITF_MBJOB_VIS,1) TO UPPER_BOUND(_ayITF_MBJOB_VIS,1) -1 DO
		IF __QUERYINTERFACE(_ayITF_MBJOB_VIS[diFor],ITF_TEMP_MBJOB_VIS) THEN
			_ayITF_MBJOB_VIS[diFor + 1]	:= _ayITF_MBJOB_VIS[diFor].LOW_SYBIL;
		ELSE
			_ayITF_MBJOB_VIS[diFor + 1] := 0;
		END_IF;	
	END_FOR;
(* Load Next 10 *)
ELSIF xLoadNext10 THEN
	IF __QUERYINTERFACE(_ayITF_MBJOB_VIS[UPPER_BOUND(_ayITF_MBJOB_VIS,1)],ITF_TEMP_MBJOB_VIS) THEN
		_ayITF_MBJOB_VIS[LOWER_BOUND(_ayITF_MBJOB_VIS,1)] := ITF_TEMP_MBJOB_VIS.LOW_SYBIL;
		FOR diFor := LOWER_BOUND(_ayITF_MBJOB_VIS,1) TO UPPER_BOUND(_ayITF_MBJOB_VIS,1) -1 DO
			IF __QUERYINTERFACE(_ayITF_MBJOB_VIS[diFor],ITF_TEMP_MBJOB_VIS) THEN
				_ayITF_MBJOB_VIS[diFor + 1]	:= _ayITF_MBJOB_VIS[diFor].LOW_SYBIL;
			ELSE
				_ayITF_MBJOB_VIS[diFor + 1] := 0;
			END_IF;	
		END_FOR;
	END_IF;
(* Load Last 10 *)
ELSIF xLoadLast10 THEN
	IF __QUERYINTERFACE(_ayITF_MBJOB_VIS[LOWER_BOUND(_ayITF_MBJOB_VIS,1)],ITF_TEMP_MBJOB_VIS) THEN
		IF __QUERYINTERFACE(_ayITF_MBJOB_VIS[LOWER_BOUND(_ayITF_MBJOB_VIS,1)].BIG_SYBIL,ITF_TEMP_SAFE) THEN
			_ayITF_MBJOB_VIS[UPPER_BOUND(_ayITF_MBJOB_VIS,1)] := ITF_TEMP_MBJOB_VIS.BIG_SYBIL;
			FOR diFor := UPPER_BOUND(_ayITF_MBJOB_VIS,1) TO LOWER_BOUND(_ayITF_MBJOB_VIS,1) + 1 BY -1 DO 
				IF __QUERYINTERFACE(_ayITF_MBJOB_VIS[diFor],ITF_TEMP_MBJOB_VIS) THEN
					ITF_TEMP_LAST_VALID  		:= _ayITF_MBJOB_VIS[diFor];
					_ayITF_MBJOB_VIS[diFor - 1]	:= _ayITF_MBJOB_VIS[diFor].BIG_SYBIL;
				ELSE
					(* Resort if new ones Inside *)
					_ayITF_MBJOB_VIS[LOWER_BOUND(_ayITF_MBJOB_VIS,1)] := ITF_TEMP_LAST_VALID;
					FOR diFor := LOWER_BOUND(_ayITF_MBJOB_VIS,1) TO UPPER_BOUND(_ayITF_MBJOB_VIS,1) -1 DO
						IF __QUERYINTERFACE(_ayITF_MBJOB_VIS[diFor],ITF_TEMP_MBJOB_VIS) THEN
							_ayITF_MBJOB_VIS[diFor + 1]	:= _ayITF_MBJOB_VIS[diFor].LOW_SYBIL;
						ELSE
							_ayITF_MBJOB_VIS[diFor + 1] := 0;
						END_IF;	
					END_FOR;					
				END_IF;	
			END_FOR;
		END_IF;
	END_IF;	
END_IF;
END_METHOD

PROPERTY IsCurrentCall : BOOL
GET
IsCurrentCall := xGetReadyCalled AND NOT xAllJobsDone;
END_GET
END_PROPERTY

PROPERTY CONFIRM_ALL_JOBS_DONE : BOOL
GET
CONFIRM_ALL_JOBS_DONE := xConfirmAllJobsDone;
END_GET
END_PROPERTY

END_FUNCTION_BLOCK

// 21 Interface/CLIENT/TCP/ITF_MB_CLIENT_TCP
INTERFACE ITF_MB_CLIENT_TCP  EXTENDS ITF_CLIENT

PROPERTY ENABLE : BOOL
GET
END_GET
END_PROPERTY

PROPERTY NODE_ID : USINT
GET
END_GET
END_PROPERTY

PROPERTY TIMEOUT : TIME
GET
END_GET
END_PROPERTY

PROPERTY READ_DELAY : TIME
GET
END_GET
END_PROPERTY

PROPERTY WRITE_DELAY : TIME
GET
END_GET
END_PROPERTY

PROPERTY IP_ADRESS : STRING(15)
GET
END_GET
END_PROPERTY

PROPERTY PORT : UINT
GET
END_GET
END_PROPERTY

PROPERTY P_fbxEnable : CtaSysConfig.ITF_DATATYPE
GET
END_GET
END_PROPERTY

PROPERTY P_fbusiNodeId : CtaSysConfig.ITF_DATATYPE
GET
END_GET
END_PROPERTY

PROPERTY P_fbtTimeOut : CtaSysConfig.ITF_DATATYPE
GET
END_GET
END_PROPERTY

PROPERTY P_fbtReadDelay : CtaSysConfig.ITF_DATATYPE
GET
END_GET
END_PROPERTY

PROPERTY P_fbtWriteDelay : CtaSysConfig.ITF_DATATYPE
GET
END_GET
END_PROPERTY

PROPERTY P_fbuiPort : CtaSysConfig.ITF_DATATYPE
GET
END_GET
END_PROPERTY

PROPERTY P_fbstIpAdress : CtaSysConfig.ITF_DATATYPE
GET
END_GET
END_PROPERTY

END_INTERFACE

// 30 Program Organization Units/FC/fcCheckIp
FUNCTION fcCheckIp : BOOL
VAR_INPUT
    stIp           : STRING[20];
END_VAR
VAR
    iFor           : INT;
    iCountPacket   : INT;
    iCountPoint    : INT;
    iCountZiffer   : INT;
    xFail          : BOOL;
END_VAR

FOR iFor := LEN(stIp) TO 0 BY -1 DO
    // Check Termination
    IF iFor = LEN(stIp) THEN
        IF stIp[iFor] <> 0 THEN 
            xFail := TRUE; // No Termination
            EXIT;       
        END_IF;
	ELSE
        // Check if Ziffer
        IF stIp[iFor] >= 48 AND stIp[iFor] <= 57 THEN    
            IF iCountZiffer < 3 THEN
                IF iCountZiffer = 0 THEN
                    IF iFor >= 2 THEN
                        IF stIp[iFor - 2] >= 50 THEN
                            // Check if Ziffer <= 5
                            IF stIp[iFor] <= 53 THEN     
                                iCountZiffer := iCountZiffer + 1;
                            ELSE
                                xFail := TRUE;  // Max is 255
                                EXIT;
                            END_IF;   
                        ELSE
                            iCountZiffer := iCountZiffer + 1;                   
						END_IF;                        
                    ELSE
                        iCountZiffer := iCountZiffer + 1;
					END_IF
                ELSIF iCountZiffer = 1 THEN
                    IF iFor <> 0 THEN
                        IF stIp[iFor - 1] = 46 THEN
                            iCountZiffer := iCountZiffer + 1;
                        // Check if next Ziffer is 2    
                        ELSIF stIp[iFor - 1] >= 50 THEN  
                            // Check if Ziffer <= 5
                            IF stIp[iFor] <= 53 THEN     
                                iCountZiffer := iCountZiffer + 1;
                            ELSE
                                xFail := TRUE;  // Max is 255
                                EXIT;
                            END_IF;    
                        END_IF;
                    ELSE
                        iCountZiffer := iCountZiffer + 1;        
					END_IF;                       
                ELSIF iCountZiffer = 2 THEN
                    IF stIp[iFor] <= 50 THEN
                        iCountZiffer := iCountZiffer + 1;
                    ELSE
                        xFail := TRUE;
                        EXIT;
					END_IF
                END_IF;    
            ELSIF iCountZiffer = 3 THEN
                xFail := TRUE; // More Then 3 Ziffers not allowed!
                EXIT;
            END_IF;
        // Check if Point
        ELSIF stIp[iFor] = 46 THEN
            IF iCountZiffer > 0 THEN
                iCountPacket := iCountPacket + 1;
                iCountPoint  := iCountPoint + 1;
                iCountZiffer := 0;
            ELSE
                xFail := TRUE; // Empty Packet not allowed!
                EXIT;
            END_IF;   
        END_IF;
    END_IF;
END_FOR;

IF xFail THEN
    fcCheckIp := FALSE;
ELSIF iCountPoint = 3 AND iCountPacket = 3 AND iCountZiffer > 0 THEN    
    fcCheckIp := TRUE;
END_IF;

END_FUNCTION

// 30 Program Organization Units/FC/fcSetInitialIPString
FUNCTION fcSetInitialIPString : BOOL
VAR_INPUT
    ITF_STRING40In : CtaSysConfig.ITF_STRING40;	
END_VAR
VAR
END_VAR

IF __QUERYINTERFACE(ITF_STRING40In,ITF_STRING40In) THEN
    IF ITF_STRING40In.proValue = '' THEN    
        ITF_STRING40In.proValue := '0.0.0.0';
    END_IF;
    fcSetInitialIPString := TRUE;
ELSE
    fcSetInitialIPString := FALSE;
END_IF;

END_FUNCTION

// 21 Interface/CLIENTMANAGER/BASE/ITF_MB_CLIENTMANAGER
INTERFACE ITF_MB_CLIENTMANAGER EXTENDS __system.IQueryInterface

PROPERTY OperationTime : LTIME
GET
END_GET
END_PROPERTY

PROPERTY ITF_BASE_CLIENT : ITF_CLIENT
GET
END_GET
END_PROPERTY

PROPERTY AY_ITF_MBCLIENT_VIS : ARRAY[0..9] OF ITF_CLIENT
GET
END_GET
END_PROPERTY

METHOD RELOAD_ARRAY
VAR_INPUT
	xInit				:	BOOL;
	xLoadNext10			:	BOOL;
	xLoadLast10			:	BOOL;
END_VAR
END_METHOD

END_INTERFACE

// 21 Interface/CLIENT/RTU/ITF_MB_CLIENT_RTU
INTERFACE ITF_MB_CLIENT_RTU  EXTENDS ITF_CLIENT

PROPERTY ENABLE : BOOL
GET
END_GET
END_PROPERTY

PROPERTY P_fbxEnable : CtaSysConfig.ITF_DATATYPE
GET
END_GET
END_PROPERTY

PROPERTY P_fbusiNodeId : CtaSysConfig.ITF_DATATYPE
GET
END_GET
END_PROPERTY

PROPERTY P_fbtTimeOut : CtaSysConfig.ITF_DATATYPE
GET
END_GET
END_PROPERTY

PROPERTY P_fbtReadDelay : CtaSysConfig.ITF_DATATYPE
GET
END_GET
END_PROPERTY

PROPERTY P_fbtWriteDelay : CtaSysConfig.ITF_DATATYPE
GET
END_GET
END_PROPERTY

PROPERTY NODE_ID : USINT
GET
END_GET
END_PROPERTY

PROPERTY TIMEOUT : TIME
GET
END_GET
END_PROPERTY

PROPERTY READ_DELAY : TIME
GET
END_GET
END_PROPERTY

PROPERTY WRITE_DELAY : TIME
GET
END_GET
END_PROPERTY

END_INTERFACE

// 30 Program Organization Units/FC/FcBytePointToWordValue
FUNCTION FcBytePointToWordValue : WORD
VAR_INPUT
	_pByte			:	POINTER TO BYTE;
END_VAR
VAR
	_pWord			:	POINTER TO Word;
END_VAR

IF _pByte <> 0 THEN
	_pWord := _pByte;
	FcBytePointToWordValue := _pWord^;
END_IF;

END_FUNCTION

// 30 Program Organization Units/FC/FcBytePointToBoolValue
FUNCTION FcBytePointToBoolValue : BOOL
VAR_INPUT
	_pByte			:	POINTER TO BYTE;
END_VAR
VAR
	_pBool			:	POINTER TO BOOL;
END_VAR

IF _pByte <> 0 THEN
	_pBool := _pByte;
	FcBytePointToBoolValue := _pBool^;
END_IF;

END_FUNCTION

// 30 Program Organization Units/FC/fcStringIPtoByteArray
FUNCTION fcStringIPtoByteArray : ARRAY[0..3] OF BYTE
VAR_INPUT
	stIP	:	STRING;
END_VAR
VAR
END_VAR

fcStringIPtoByteArray	:= IoDrvEthernet.UDINT_TO_IPARRAY(IoDrvEthernet.IPSTRING_TO_UDINT(stIp));

END_FUNCTION

// 30 Program Organization Units/CLIENTMANAGER/TCP/FB_MB_CLIENTMANAGER_TCP
{attribute 'no_assign'}
FUNCTION_BLOCK FB_MB_CLIENTMANAGER_TCP EXTENDS FB_MB_CLIENTMANAGER IMPLEMENTS ITF_MB_CLIENTMANAGER_TCP
VAR_OUTPUT
END_VAR
VAR
	Client								:	ModbusFB.ClientTCP;

	_TEMP_MBU_CLIENT_TCP				:	ITF_MB_CLIENT_TCP;
	
	fbReadCoilsFc01						:	ModbusFB.ClientRequestReadCoils;
	fbReadDiscreteInputsFc02			:	ModbusFB.ClientRequestReadDiscreteInputs;
	fbReadHoldingRegistersFc03			:	ModbusFB.ClientRequestReadHoldingRegisters;
	fbReadInputRegistersFc04			:	ModbusFB.ClientRequestReadInputRegisters;
	fbWriteSingleCoilFc05				:	ModbusFB.ClientRequestWriteSingleCoil;
	fbWriteSingleRegisterFc06			:	ModbusFB.ClientRequestWriteSingleRegister;
	fbWriteMultipleCoilsFc15			:	ModbusFB.ClientRequestWriteMultipleCoils;
	fbWriteMultipleRegistersFc16		:	ModbusFB.ClientRequestWriteMultipleRegisters;
	
END_VAR

SUPER^();
(* Check if one is allready Working *)
IF NOT xIsWorking THEN
	(* Get Client Ready *)
	IF __QUERYINTERFACE(_TEMP_MBU_CLIENT,_TEMP_MBU_CLIENT) THEN
		xIsWorking 		:= TRUE;	
		xErrorHappen	:= FALSE;
		eErrorID		:= ModbusFB.Error.OK;
		eExeptionCode	:= ModbusFB.ExceptionCodes.RESPONSE_SUCCESS;		
	(* Get Base Client Ready *)
	ELSIF __QUERYINTERFACE(_BASE_MBU_CLIENT,_TEMP_MBU_CLIENT) THEN
		xIsWorking 		:= TRUE;
		xErrorHappen	:= FALSE;
		eErrorID		:= ModbusFB.Error.OK;
		eExeptionCode	:= ModbusFB.ExceptionCodes.RESPONSE_SUCCESS;
		ltTime 			:= fbTimeStop.Stop();
		fbTimeStop.Start();
	END_IF;
END_IF;
(* Check if is running *)
IF xIsWorking THEN
	IF __QUERYINTERFACE(_TEMP_MBU_CLIENT,_TEMP_MBU_CLIENT) THEN	
		(* Wait until no Execute *)		
		IF 	NOT	fbReadCoilsFc01.xExecute				AND
			NOT	fbReadDiscreteInputsFc02.xExecute	    AND
			NOT	fbReadHoldingRegistersFc03.xExecute     AND
			NOT	fbReadInputRegistersFc04.xExecute	    AND
			NOT	fbWriteSingleCoilFc05.xExecute		    AND
			NOT	fbWriteSingleRegisterFc06.xExecute	    AND
			NOT	fbWriteMultipleCoilsFc15.xExecute	    AND
			NOT	fbWriteMultipleRegistersFc16.xExecute	THEN
			(* Connect *)
			IF NOT Client.xConnected THEN
				(* Get Type of Port *) 
				IF __QUERYINTERFACE(_TEMP_MBU_CLIENT,_TEMP_MBU_CLIENT_TCP) THEN
					(* Check if Enabled *)
					IF _TEMP_MBU_CLIENT_TCP.ENABLE AND _TEMP_MBU_CLIENT_TCP.COUNT > 0 THEN
						_TEMP_MBU_CLIENT.GET_READY();
						IF fcCheckIp(_TEMP_MBU_CLIENT_TCP.IP_ADRESS) THEN
							Client.uiPort 	:= _TEMP_MBU_CLIENT_TCP.PORT;
							Client.aIPaddr 	:= fcStringIPtoByteArray(_TEMP_MBU_CLIENT_TCP.IP_ADRESS);
							Client.xConnect	:= TRUE;
							usiNodeId 		:= _TEMP_MBU_CLIENT_TCP.NODE_ID;
							tTimeOut		:= _TEMP_MBU_CLIENT_TCP.TIMEOUT;
							tReadDelay		:= _TEMP_MBU_CLIENT_TCP.READ_DELAY;
							tWriteDelay	 	:= _TEMP_MBU_CLIENT_TCP.WRITE_DELAY;
						ELSE
							xAbort := TRUE;
						END_IF;
					ELSE
						xAbort		:= TRUE;
					END_IF;
				ELSE
					xAbort := TRUE;
				END_IF;
			END_IF;
			(* Check if Connected *)
			IF Client.xConnected AND NOT xAbort THEN
				(* Get Job *)
				IF NOT xTrig THEN
					xTrig := _TEMP_MBU_CLIENT.GET_NEXT_JOB(_byMbFunction => _byMbFunction,_wMbAdress => _wMbAdress,_pByte => _pByte,_wQuantity => _wQuantity);
				END_IF;
				
				(* Delay Function *)
				actDelays();
				
				(* Execute Function *)
				actExecuteFunction();
				
				(* Resett Timer *)
				IF tonDelay.Q THEN
					tonDelay(IN := FALSE);
					xTrig := FALSE;
				END_IF;
			END_IF;
		ELSE
			(* Check Busy *)
			actCheckBusy();					
		END_IF;
		(* Get Errors *)
		actGetError();
		(* Check if All Job as Done *)
		IF _TEMP_MBU_CLIENT.AllJobsDone OR xAbort THEN
			(* Wait until no Execute *)		
			IF 	NOT	fbReadCoilsFc01.xExecute				AND
				NOT	fbReadDiscreteInputsFc02.xExecute	    AND
				NOT	fbReadHoldingRegistersFc03.xExecute     AND
				NOT	fbReadInputRegistersFc04.xExecute	    AND
				NOT	fbWriteSingleCoilFc05.xExecute		    AND
				NOT	fbWriteSingleRegisterFc06.xExecute	    AND
				NOT	fbWriteMultipleCoilsFc15.xExecute	    AND
				NOT	fbWriteMultipleRegistersFc16.xExecute	THEN
				_TEMP_MBU_CLIENT.CALL_AFTER_LAST_JOB_DONE();
				(* Set Error if Job > 0 *)
				IF _TEMP_MBU_CLIENT.COUNT > 0 THEN
					_TEMP_MBU_CLIENT.ERROR			:= xErrorHappen;
					_TEMP_MBU_CLIENT.ERROR_ID		:= eErrorID;
					_TEMP_MBU_CLIENT.EXEPTION_CODE	:= eExeptionCode;
				END_IF;
				_TEMP_MBU_CLIENT 				:= _TEMP_MBU_CLIENT.LOW_SYBIL;
				xIsWorking						:= FALSE;
				xAbort							:= FALSE;
				Client.xConnect					:= FALSE;
			END_IF;
		END_IF;
	END_IF;
END_IF;

(* Call Functions *)
actCallFunctions();

(* Resett Client on Error *)
IF Client.xError THEN
	Client.xConnect := FALSE;
END_IF
(* Call Client *)
Client();

ACTION actGetError:
(* Client Error *)
IF Client.xError THEN
	xErrorHappen 	:= Client.xError;
	eErrorID		:= Client.eErrorID;
	eExeptionCode	:= ModbusFB.ExceptionCodes.ACKNOWLEDGE;
	xAbort			:= TRUE;
END_IF;
(* Read Coils Fc01 Error *)
IF fbReadCoilsFc01.xError AND NOT xErrorHappen THEN
	xErrorHappen 	:= fbReadCoilsFc01.xError;
	eErrorID		:= fbReadCoilsFc01.eErrorID;
	eExeptionCode	:= fbReadCoilsFc01.eException;
END_IF;
(* Read Discrete Inputs Fc02 Error *)
IF fbReadDiscreteInputsFc02.xError AND NOT xErrorHappen THEN
	xErrorHappen 	:= fbReadDiscreteInputsFc02.xError;
	eErrorID		:= fbReadDiscreteInputsFc02.eErrorID;
	eExeptionCode	:= fbReadDiscreteInputsFc02.eException;
END_IF;
(* Read Holding Registers Fc03 Error *)
IF fbReadHoldingRegistersFc03.xError AND NOT xErrorHappen THEN
	xErrorHappen 	:= fbReadHoldingRegistersFc03.xError;
	eErrorID		:= fbReadHoldingRegistersFc03.eErrorID;
	eExeptionCode	:= fbReadHoldingRegistersFc03.eException;
END_IF;
(* Read Input Registers Fc04 Error *)
IF fbReadInputRegistersFc04.xError AND NOT xErrorHappen THEN
	xErrorHappen 	:= fbReadInputRegistersFc04.xError;
	eErrorID		:= fbReadInputRegistersFc04.eErrorID;
	eExeptionCode	:= fbReadInputRegistersFc04.eException;
END_IF;
(* Write Single Coil Fc05 Error *)
IF fbWriteSingleCoilFc05.xError AND NOT xErrorHappen THEN
	xErrorHappen 	:= fbWriteSingleCoilFc05.xError;
	eErrorID		:= fbWriteSingleCoilFc05.eErrorID;
	eExeptionCode	:= fbWriteSingleCoilFc05.eException;
END_IF;
(* Write Single Register Fc06 Error *)
IF fbWriteSingleRegisterFc06.xError AND NOT xErrorHappen THEN
	xErrorHappen 	:= fbWriteSingleRegisterFc06.xError;
	eErrorID		:= fbWriteSingleRegisterFc06.eErrorID;
	eExeptionCode	:= fbWriteSingleRegisterFc06.eException;
END_IF;		
(* Write Multiple Coils Fc15 Error *)
IF fbWriteMultipleCoilsFc15.xError AND NOT xErrorHappen THEN
	xErrorHappen 	:= fbWriteMultipleCoilsFc15.xError;
	eErrorID		:= fbWriteMultipleCoilsFc15.eErrorID;
	eExeptionCode	:= fbWriteMultipleCoilsFc15.eException;
END_IF;
(* Write Multiple Registers Fc16 Error *)
IF fbWriteMultipleRegistersFc16.xError AND NOT xErrorHappen THEN
	xErrorHappen 	:= fbWriteMultipleRegistersFc16.xError;
	eErrorID		:= fbWriteMultipleRegistersFc16.eErrorID;
	eExeptionCode	:= fbWriteMultipleRegistersFc16.eException;
END_IF;
END_ACTION

ACTION actCheckBusy:
(* Reset after Busy *)
fbReadCoilsFc01.xExecute				:= fbReadCoilsFc01.xBusy				;
fbReadDiscreteInputsFc02.xExecute	    := fbReadDiscreteInputsFc02.xBusy		;
fbReadHoldingRegistersFc03.xExecute     := fbReadHoldingRegistersFc03.xBusy		;
fbReadInputRegistersFc04.xExecute	    := fbReadInputRegistersFc04.xBusy		;
fbWriteSingleCoilFc05.xExecute		    := fbWriteSingleCoilFc05.xBusy			;
fbWriteSingleRegisterFc06.xExecute	    := fbWriteSingleRegisterFc06.xBusy		;
fbWriteMultipleCoilsFc15.xExecute	    := fbWriteMultipleCoilsFc15.xBusy		;
fbWriteMultipleRegistersFc16.xExecute   := fbWriteMultipleRegistersFc16.xBusy	;
END_ACTION

ACTION actExecuteFunction:
(* Read Coils *)
IF _byMbFunction = 01 THEN
	fbReadCoilsFc01.udiReplyTimeout					:= TO_UDINT(tTimeOut) * 1000; 
	fbReadCoilsFc01.udiTimeOut						:= 1000000;
	fbReadCoilsFc01.uiUnitId						:= usiNodeId;
	fbReadCoilsFc01.uiStartItem 					:= TO_UINT(_wMbAdress);
	fbReadCoilsFc01.pData 							:= _pByte;
	fbReadCoilsFc01.uiQuantity						:= TO_UINT(_wQuantity);
	fbReadCoilsFc01.xExecute						:= tonDelay.Q;
(* Read Discret Inputs *)                       	
ELSIF _byMbFunction = 02 THEN                   	
	fbReadDiscreteInputsFc02.udiReplyTimeout		:= TO_UDINT(tTimeOut) * 1000; 
	fbReadDiscreteInputsFc02.udiTimeOut				:= 1000000;
	fbReadDiscreteInputsFc02.uiUnitId				:= usiNodeId;
	fbReadDiscreteInputsFc02.uiStartItem			:= TO_UINT(_wMbAdress);
	fbReadDiscreteInputsFc02.pData 					:= _pByte;
	fbReadDiscreteInputsFc02.uiQuantity				:= TO_UINT(_wQuantity);
	fbReadDiscreteInputsFc02.xExecute				:= tonDelay.Q;
(* Read Holding Registers *)                		
ELSIF _byMbFunction = 03 THEN                   	
	fbReadHoldingRegistersFc03.udiReplyTimeout		:= TO_UDINT(tTimeOut) * 1000; 
	fbReadHoldingRegistersFc03.udiTimeOut			:= 1000000;
	fbReadHoldingRegistersFc03.uiUnitId				:= usiNodeId;          	
	fbReadHoldingRegistersFc03.uiStartItem			:= TO_UINT(_wMbAdress);
	fbReadHoldingRegistersFc03.pData 				:= _pByte;
	fbReadHoldingRegistersFc03.uiQuantity			:= TO_UINT(_wQuantity);
	fbReadHoldingRegistersFc03.xExecute				:= tonDelay.Q;			
(* Read Input Registers *)	                		
ELSIF _byMbFunction = 04 THEN                   	
	fbReadInputRegistersFc04.udiReplyTimeout		:= TO_UDINT(tTimeOut) * 1000; 
	fbReadInputRegistersFc04.udiTimeOut				:= 1000000;
	fbReadInputRegistersFc04.uiUnitId				:= usiNodeId;               	
	fbReadInputRegistersFc04.uiStartItem 			:= TO_UINT(_wMbAdress);
	fbReadInputRegistersFc04.pData 					:= _pByte;
	fbReadInputRegistersFc04.uiQuantity				:= TO_UINT(_wQuantity);
	fbReadInputRegistersFc04.xExecute				:= tonDelay.Q;			
(* Write Single Coil *)	                    		
ELSIF _byMbFunction = 05 THEN                   	
	fbWriteSingleCoilFc05.udiReplyTimeout			:= TO_UDINT(tTimeOut) * 1000; 
	fbWriteSingleCoilFc05.udiTimeOut				:= 1000000;
	fbWriteSingleCoilFc05.uiUnitId					:= usiNodeId;            	
	fbWriteSingleCoilFc05.uiItem 					:= TO_UINT(_wMbAdress);
	fbWriteSingleCoilFc05.xValue 					:= FcBytePointToBoolValue(_pByte);
	fbWriteSingleCoilFc05.xExecute					:= tonDelay.Q;		
(* Write Single Register *)                 		
ELSIF _byMbFunction = 06 THEN                   	
	fbWriteSingleRegisterFc06.udiReplyTimeout		:= TO_UDINT(tTimeOut) * 1000;    
	fbWriteSingleRegisterFc06.udiTimeOut			:= 1000000; 
	fbWriteSingleRegisterFc06.uiUnitId				:= usiNodeId;           	
	fbWriteSingleRegisterFc06.uiItem	  			:= TO_UINT(_wMbAdress);
	fbWriteSingleRegisterFc06.uiValue 				:= FcBytePointToWordValue(_pByte);
	fbWriteSingleRegisterFc06.xExecute				:= tonDelay.Q;		
(* Write Multiple Coils *)		            		
ELSIF _byMbFunction = 15 THEN                   	
	fbWriteMultipleCoilsFc15.udiReplyTimeout		:= TO_UDINT(tTimeOut) * 1000;
	fbWriteMultipleCoilsFc15.udiTimeOut				:= 1000000;
	fbWriteMultipleCoilsFc15.uiUnitId				:= usiNodeId;              	
	fbWriteMultipleCoilsFc15.uiStartItem 			:= TO_UINT(_wMbAdress);
	fbWriteMultipleCoilsFc15.pData 					:= _pByte;
	fbWriteMultipleCoilsFc15.uiQuantity				:= TO_UINT(_wQuantity);
	fbWriteMultipleCoilsFc15.xExecute				:= tonDelay.Q;
(* Write Multiple Registers *)                  	
ELSIF _byMbFunction = 16 THEN                   	
	fbWriteMultipleRegistersFc16.udiReplyTimeout	:= TO_UDINT(tTimeOut) * 1000; 
	fbWriteMultipleRegistersFc16.udiTimeOut			:= 1000000;
	fbWriteMultipleRegistersFc16.uiUnitId			:= usiNodeId;    
	fbWriteMultipleRegistersFc16.uiStartItem 		:= TO_UINT(_wMbAdress);
	fbWriteMultipleRegistersFc16.pData 				:= _pByte;
	fbWriteMultipleRegistersFc16.uiQuantity			:= TO_UINT(_wQuantity);
	fbWriteMultipleRegistersFc16.xExecute			:= tonDelay.Q;	
END_IF;
END_ACTION

ACTION actDelays:
(* Delay Read *)
IF _byMbFunction <= 04 THEN
	tonDelay(IN := xTrig,PT := tReadDelay);
(* Delay Write Single *)
ELSIF _byMbFunction >= 5 AND _byMbFunction <= 6 THEN
	tonDelay(IN := xTrig,PT := tWriteDelay); 
(* Delay Write Multiple *)
ELSIF _byMbFunction >= 15 AND _byMbFunction <= 16 THEN
	tonDelay(IN := xTrig,PT := tWriteDelay); 
ELSE 
	tonDelay(IN := xTrig,PT := T#0MS);
END_IF;
END_ACTION

ACTION actCallFunctions:
(* Call *)
fbReadCoilsFc01(				rClient := client);				
fbReadDiscreteInputsFc02(		rClient := Client);  
fbReadHoldingRegistersFc03(		rClient := Client);
fbReadInputRegistersFc04(		rClient := Client);	  
fbWriteSingleCoilFc05(			rClient := Client);	  
fbWriteSingleRegisterFc06(		rClient := Client);  
fbWriteMultipleCoilsFc15(		rClient := Client);  
fbWriteMultipleRegistersFc16(	rClient := Client);
END_ACTION

END_FUNCTION_BLOCK

// 30 Program Organization Units/CLIENTMANAGER/BASE/FB_MB_CLIENTMANAGER
{attribute 'no_assign'}
FUNCTION_BLOCK FB_MB_CLIENTMANAGER EXTENDS CtaAppBmk.fbBMK IMPLEMENTS ITF_MB_CLIENTMANAGER
VAR_OUTPUT
END_VAR
VAR
	_BASE_MBU_CLIENT					:	ITF_CLIENT;
	_TEMP_REG_CLIENT					:	ITF_CLIENT;
	_TEMP_MBU_CLIENT					:	ITF_CLIENT;		
	_COUNT								:	UINT;
	
	xIsWorking							:	BOOL;
	xTrig								:	BOOL;
	xAbort								:	BOOL;
	xErrorHappen						:	BOOL;
	eErrorID							:	ModbusFB.Error;
	eExeptionCode						:	ModbusFB.ExceptionCodes;
	
	usiNodeId							:	USINT;
	
	tTimeOut							:	TIME;
	tReadDelay							:	TIME;
	tWriteDelay							:	TIME;
	tonDelay							:	Standard.TON;
	_byMbFunction						:	BYTE;
	_wMbAdress							:	WORD;
	_pByte								:	POINTER TO BYTE;
	_wQuantity							:	WORD;	
	                					
	fbTimeStop							:	CtaAppTime.fbTimeMeasurement;
	ltTime								:	LTIME;

	_ayITF_MBCLIENT_VIS					:	ARRAY[0..9] OF ITF_CLIENT;
END_VAR

PROPERTY ITF_BASE_CLIENT : ITF_CLIENT
GET
END_GET
END_PROPERTY

METHOD ADD_MODBUS_CLIENT
VAR_INPUT
	ITF_CLIENT_IN	:	ITF_CLIENT;
END_VAR
IF NOT CHECK_IF_EXIST(ITF_CLIENT_IN) THEN
	IF __QUERYINTERFACE(ITF_CLIENT_IN,ITF_CLIENT_IN) THEN
		IF __QUERYINTERFACE(_BASE_MBU_CLIENT,_BASE_MBU_CLIENT) THEN
			IF __QUERYINTERFACE(_TEMP_REG_CLIENT,_TEMP_REG_CLIENT) THEN
				_TEMP_REG_CLIENT.LOW_SYBIL := ITF_CLIENT_IN;
				_TEMP_REG_CLIENT := ITF_CLIENT_IN;
			ELSE
				_BASE_MBU_CLIENT.LOW_SYBIL := ITF_CLIENT_IN;
				_TEMP_REG_CLIENT := ITF_CLIENT_IN;		
			END_IF;		
		ELSE
			_BASE_MBU_CLIENT := ITF_CLIENT_IN;
		END_IF;
		THIS^.RELOAD_ARRAY(TRUE,FALSE,FALSE);
		_COUNT := _COUNT + 1;
	END_IF;
END_IF;
END_METHOD

METHOD CHECK_IF_EXIST : BOOL
VAR_INPUT
	ITF_CLIENT_IN	:	ITF_CLIENT;
END_VAR
VAR
	ITF_CLIENT_TEMP	:	ITF_CLIENT;
END_VAR
IF __QUERYINTERFACE(_BASE_MBU_CLIENT,ITF_CLIENT_TEMP) THEN
	REPEAT
		IF __QUERYINTERFACE(ITF_CLIENT_TEMP,ITF_CLIENT_TEMP) THEN
			IF ITF_CLIENT_IN = ITF_CLIENT_TEMP THEN
				CHECK_IF_EXIST := TRUE;
			END_IF
			ITF_CLIENT_TEMP := ITF_CLIENT_TEMP.LOW_SYBIL;
		ELSE
			ITF_CLIENT_TEMP := 0;
		END_IF;
	UNTIL ITF_CLIENT_TEMP = 0 
	END_REPEAT;
END_IF
END_METHOD

METHOD RELOAD_ARRAY
VAR_INPUT
	xInit	: BOOL;
	xLoadNext10	: BOOL;
	xLoadLast10	: BOOL;
END_VAR
VAR
	diFor				:	DINT;
	ITF_TEMP_CLIENT_VIS	:	ITF_CLIENT;
	ITF_TEMP_SAFE		:	ITF_CLIENT;
	ITF_TEMP_LAST_VALID	:	ITF_CLIENT;
END_VAR
(* Init Array *)
IF xInit THEN
	_ayITF_MBCLIENT_VIS[LOWER_BOUND(_ayITF_MBCLIENT_VIS,1)] := _BASE_MBU_CLIENT;
	FOR diFor := LOWER_BOUND(_ayITF_MBCLIENT_VIS,1) TO UPPER_BOUND(_ayITF_MBCLIENT_VIS,1) -1 DO
		IF __QUERYINTERFACE(_ayITF_MBCLIENT_VIS[diFor],ITF_TEMP_CLIENT_VIS) THEN
			_ayITF_MBCLIENT_VIS[diFor + 1]	:= _ayITF_MBCLIENT_VIS[diFor].LOW_SYBIL;
		ELSE
			_ayITF_MBCLIENT_VIS[diFor + 1] := 0;
		END_IF;	
	END_FOR;
(* Load Next 10 *)
ELSIF xLoadNext10 THEN
	IF __QUERYINTERFACE(_ayITF_MBCLIENT_VIS[UPPER_BOUND(_ayITF_MBCLIENT_VIS,1)],ITF_TEMP_CLIENT_VIS) THEN
		_ayITF_MBCLIENT_VIS[LOWER_BOUND(_ayITF_MBCLIENT_VIS,1)] := ITF_TEMP_CLIENT_VIS.LOW_SYBIL;
		FOR diFor := LOWER_BOUND(_ayITF_MBCLIENT_VIS,1) TO UPPER_BOUND(_ayITF_MBCLIENT_VIS,1) -1 DO
			IF __QUERYINTERFACE(_ayITF_MBCLIENT_VIS[diFor],ITF_TEMP_CLIENT_VIS) THEN
				_ayITF_MBCLIENT_VIS[diFor + 1]	:= _ayITF_MBCLIENT_VIS[diFor].LOW_SYBIL;
			ELSE
				_ayITF_MBCLIENT_VIS[diFor + 1] := 0;
			END_IF;	
		END_FOR;
	END_IF;
(* Load Last 10 *)
ELSIF xLoadLast10 THEN
	IF __QUERYINTERFACE(_ayITF_MBCLIENT_VIS[LOWER_BOUND(_ayITF_MBCLIENT_VIS,1)],ITF_TEMP_CLIENT_VIS) THEN
		IF __QUERYINTERFACE(_ayITF_MBCLIENT_VIS[LOWER_BOUND(_ayITF_MBCLIENT_VIS,1)].BIG_SYBIL,ITF_TEMP_SAFE) THEN
			_ayITF_MBCLIENT_VIS[UPPER_BOUND(_ayITF_MBCLIENT_VIS,1)] := ITF_TEMP_CLIENT_VIS.BIG_SYBIL;
			FOR diFor := UPPER_BOUND(_ayITF_MBCLIENT_VIS,1) TO LOWER_BOUND(_ayITF_MBCLIENT_VIS,1) + 1 BY -1 DO 
				IF __QUERYINTERFACE(_ayITF_MBCLIENT_VIS[diFor],ITF_TEMP_CLIENT_VIS) THEN
					ITF_TEMP_LAST_VALID  			:= _ayITF_MBCLIENT_VIS[diFor];
					_ayITF_MBCLIENT_VIS[diFor - 1]	:= _ayITF_MBCLIENT_VIS[diFor].BIG_SYBIL;
				ELSE
					(* Resort if new ones Inside *)
					_ayITF_MBCLIENT_VIS[LOWER_BOUND(_ayITF_MBCLIENT_VIS,1)] := ITF_TEMP_LAST_VALID;
					FOR diFor := LOWER_BOUND(_ayITF_MBCLIENT_VIS,1) TO UPPER_BOUND(_ayITF_MBCLIENT_VIS,1) -1 DO
						IF __QUERYINTERFACE(_ayITF_MBCLIENT_VIS[diFor],ITF_TEMP_CLIENT_VIS) THEN
							_ayITF_MBCLIENT_VIS[diFor + 1]	:= _ayITF_MBCLIENT_VIS[diFor].LOW_SYBIL;
						ELSE
							_ayITF_MBCLIENT_VIS[diFor + 1] := 0;
						END_IF;	
					END_FOR;					
				END_IF;	
			END_FOR;
		END_IF;
	END_IF;	
END_IF;
END_METHOD

PROPERTY AY_ITF_MBCLIENT_VIS : ARRAY [0..9] OF ITF_CLIENT
GET
AY_ITF_MBCLIENT_VIS := _ayITF_MBCLIENT_VIS;
END_GET
END_PROPERTY

PROPERTY OperationTime : LTIME
GET
OperationTime := ltTime;
END_GET
END_PROPERTY

END_FUNCTION_BLOCK

// 21 Interface/CLIENTMANAGER/TCP/ITF_MB_CLIENTMANAGER_TCP
INTERFACE ITF_MB_CLIENTMANAGER_TCP EXTENDS ITF_MB_CLIENTMANAGER

END_INTERFACE

// 30 Program Organization Units/CLIENTMANAGER/RTU/FB_MB_CLIENTMANAGER_RTU
{attribute 'no_assign'}
FUNCTION_BLOCK FB_MB_CLIENTMANAGER_RTU EXTENDS FB_MB_CLIENTMANAGER IMPLEMENTS ITF_MB_CLIENTMANAGER_RTU
VAR_OUTPUT
END_VAR
VAR
	Client								:	ModbusFB.ClientSerial;
	
	_TEMP_MBU_CLIENT_RTU				:	ITF_MB_CLIENT_RTU;
	
	fbReadCoilsFc01						:	ModbusFB.ClientRequestReadCoils;
	fbReadDiscreteInputsFc02			:	ModbusFB.ClientRequestReadDiscreteInputs;
	fbReadHoldingRegistersFc03			:	ModbusFB.ClientRequestReadHoldingRegisters;
	fbReadInputRegistersFc04			:	ModbusFB.ClientRequestReadInputRegisters;
	fbWriteSingleCoilFc05				:	ModbusFB.ClientRequestWriteSingleCoil;
	fbWriteSingleRegisterFc06			:	ModbusFB.ClientRequestWriteSingleRegister;
	fbWriteMultipleCoilsFc15			:	ModbusFB.ClientRequestWriteMultipleCoils;
	fbWriteMultipleRegistersFc16		:	ModbusFB.ClientRequestWriteMultipleRegisters;
	
	(*Config File *)
	fbConfigFile						:	CtaSysConfig.fbConfigFile;
	scParameter                	 		: 	scSerialPortParameter;
END_VAR

SUPER^();
(* Config *)
actConfig();
(* Check if one is allready Working *)
IF NOT xIsWorking THEN
	(* Get Client Ready *)
	IF __QUERYINTERFACE(_TEMP_MBU_CLIENT,_TEMP_MBU_CLIENT) THEN
		xIsWorking := TRUE;	
		xErrorHappen	:= FALSE;
		eErrorID		:= ModbusFB.Error.OK;
		eExeptionCode	:= ModbusFB.ExceptionCodes.RESPONSE_SUCCESS;	
	(* Get Base Client Ready *)
	ELSIF __QUERYINTERFACE(_BASE_MBU_CLIENT,_TEMP_MBU_CLIENT) THEN
		xIsWorking 		:= TRUE;
		xErrorHappen	:= FALSE;
		eErrorID		:= ModbusFB.Error.OK;
		eExeptionCode	:= ModbusFB.ExceptionCodes.RESPONSE_SUCCESS;
		ltTime := fbTimeStop.Stop();
		fbTimeStop.Start();
	END_IF;
END_IF;
(* Check if is running *)
IF xIsWorking THEN
	IF __QUERYINTERFACE(_TEMP_MBU_CLIENT,_TEMP_MBU_CLIENT) THEN	
		(* Wait until no Execute *)		
		IF 	NOT	fbReadCoilsFc01.xExecute				AND
			NOT	fbReadDiscreteInputsFc02.xExecute	    AND
			NOT	fbReadHoldingRegistersFc03.xExecute     AND
			NOT	fbReadInputRegistersFc04.xExecute	    AND
			NOT	fbWriteSingleCoilFc05.xExecute		    AND
			NOT	fbWriteSingleRegisterFc06.xExecute	    AND
			NOT	fbWriteMultipleCoilsFc15.xExecute	    AND
			NOT	fbWriteMultipleRegistersFc16.xExecute	THEN
			(* Get Type of Port *) 
			IF __QUERYINTERFACE(_TEMP_MBU_CLIENT,_TEMP_MBU_CLIENT_RTU) THEN
				(* Check if Enabled *)
				IF _TEMP_MBU_CLIENT_RTU.ENABLE AND _TEMP_MBU_CLIENT_RTU.COUNT > 0 THEN
					_TEMP_MBU_CLIENT.GET_READY();
					(* Connect *)
					IF NOT Client.xConnected THEN
						Client.xConnect		:= TRUE;
						Client.iPort		:= scParameter.fbenPort.proValue;
						Client.dwBaudrate	:= scParameter.fbdwBaudrate.proValue;
						Client.byDataBits	:= scParameter.fbbyDataBits.proValue;
						Client.eParity		:= scParameter.fbenParity.proValue;
						Client.eStopBits	:= scParameter.fbenStopBits.proValue;
						Client.eDTRcontrol	:= scParameter.fbenDTRControl.proValue;
						Client.eRTScontrol	:= scParameter.fbenRTSControl.proValue;
						IF scParameter.fbxRtuAscii.proValue THEN
							Client.eRtuAscii	:= ModbusFB.RtuAscii.ASCII;
						ELSE
							Client.eRtuAscii	:= ModbusFB.RtuAscii.RTU;
						END_IF
					END_IF;
					usiNodeId 			:= _TEMP_MBU_CLIENT_RTU.NODE_ID;
					tTimeOut			:= _TEMP_MBU_CLIENT_RTU.TIMEOUT;
					tReadDelay			:= _TEMP_MBU_CLIENT_RTU.READ_DELAY;
					tWriteDelay	 		:= _TEMP_MBU_CLIENT_RTU.WRITE_DELAY;
				ELSE
					xAbort		:= TRUE;
				END_IF;
			ELSE
				xAbort		:= TRUE;				
			END_IF;
			(* Check if Connected *)
			IF Client.xConnected AND NOT xAbort THEN
				(* Get Job *)
				IF NOT xTrig THEN
					xTrig := _TEMP_MBU_CLIENT.GET_NEXT_JOB(_byMbFunction => _byMbFunction,_wMbAdress => _wMbAdress,_pByte => _pByte,_wQuantity => _wQuantity);
				END_IF;
				
				(* Delay Function *)
				actDelays();
				
				(* Execute Function *)
				actExecuteFunction();
				
				(* Resett Timer *)
				IF tonDelay.Q THEN
					tonDelay(IN := FALSE);
					xTrig := FALSE;
				END_IF;
			END_IF;
		ELSE
			(* Check Busy *)
			actCheckBusy();					
		END_IF;
		(* Get Errors *)
		actGetError();
		(* Check if All Job as Done *)
		IF _TEMP_MBU_CLIENT.AllJobsDone OR xAbort THEN
			(* Wait until no Execute *)		
			IF 	NOT	fbReadCoilsFc01.xExecute				AND
				NOT	fbReadDiscreteInputsFc02.xExecute	    AND
				NOT	fbReadHoldingRegistersFc03.xExecute     AND
				NOT	fbReadInputRegistersFc04.xExecute	    AND
				NOT	fbWriteSingleCoilFc05.xExecute		    AND
				NOT	fbWriteSingleRegisterFc06.xExecute	    AND
				NOT	fbWriteMultipleCoilsFc15.xExecute	    AND
				NOT	fbWriteMultipleRegistersFc16.xExecute	THEN
				_TEMP_MBU_CLIENT.CALL_AFTER_LAST_JOB_DONE();
				_TEMP_MBU_CLIENT.ERROR			:= xErrorHappen;
				_TEMP_MBU_CLIENT.ERROR_ID		:= eErrorID;
				_TEMP_MBU_CLIENT.EXEPTION_CODE	:= eExeptionCode;
				_TEMP_MBU_CLIENT 				:= _TEMP_MBU_CLIENT.LOW_SYBIL;
				xIsWorking						:= FALSE;
				xAbort							:= FALSE;
			END_IF;
		END_IF;
	END_IF;
END_IF;

(* Call Functions *)
actCallFunctions();

(* Resett Client on Error *)
IF Client.xError THEN
	Client.xConnect := FALSE;
END_IF
(* Call Client *)
Client();

ACTION actConfig:
fbConfigFile();		
scParameter.fbenPort			(_usiParaNr := 1,itfConfigFb := fbconfigFile , _MinInit :=    0,_MaxInit :=    10);
scParameter.fbdwBaudrate		(_usiParaNr := 2,itfConfigFb := fbconfigFile , _MinInit := 4800,_MaxInit := 115200);
scParameter.fbbyDataBits		(_usiParaNr := 3,itfConfigFb := fbconfigFile , _MinInit :=    0,_MaxInit :=     8);
scParameter.fbenParity			(_usiParaNr := 4,itfConfigFb := fbconfigFile , _MinInit :=    0,_MaxInit :=     2);
scParameter.fbenStopBits		(_usiParaNr := 5,itfConfigFb := fbconfigFile , _MinInit :=    1,_MaxInit :=     3);
scParameter.fbenDTRControl		(_usiParaNr := 6,itfConfigFb := fbconfigFile , _MinInit :=    0,_MaxInit :=     2);
scParameter.fbenRTSControl		(_usiParaNr := 7,itfConfigFb := fbconfigFile , _MinInit :=    0,_MaxInit :=     2);
scParameter.fbxRtuAscii			(_usiParaNr := 8,itfConfigFb := fbconfigFile 								 	);

(* Handle on Change *)
IF scParameter.fbenPort.proStateChanged			OR
   scParameter.fbdwBaudrate.proStateChanged	    OR
   scParameter.fbbyDataBits.proStateChanged	    OR
   scParameter.fbenParity.proStateChanged		OR
   scParameter.fbenStopBits.proStateChanged	    OR
   scParameter.fbenDTRControl.proStateChanged	OR
   scParameter.fbenRTSControl.proStateChanged	OR
   scParameter.fbxRtuAscii.proStateChanged		THEN
   Client.xConnect := FALSE;
END_IF;
END_ACTION

ACTION actGetError:
(* Client Error *)
IF Client.xError THEN
	xErrorHappen 	:= Client.xError;
	eErrorID		:= Client.eErrorID;
	eExeptionCode	:= ModbusFB.ExceptionCodes.ACKNOWLEDGE;
	xAbort			:= TRUE;
END_IF;
(* Read Coils Fc01 Error *)
IF fbReadCoilsFc01.xError AND NOT xErrorHappen THEN
	xErrorHappen 	:= fbReadCoilsFc01.xError;
	eErrorID		:= fbReadCoilsFc01.eErrorID;
	eExeptionCode	:= fbReadCoilsFc01.eException;
END_IF;
(* Read Discrete Inputs Fc02 Error *)
IF fbReadDiscreteInputsFc02.xError AND NOT xErrorHappen THEN
	xErrorHappen 	:= fbReadDiscreteInputsFc02.xError;
	eErrorID		:= fbReadDiscreteInputsFc02.eErrorID;
	eExeptionCode	:= fbReadDiscreteInputsFc02.eException;
END_IF;
(* Read Holding Registers Fc03 Error *)
IF fbReadHoldingRegistersFc03.xError AND NOT xErrorHappen THEN
	xErrorHappen 	:= fbReadHoldingRegistersFc03.xError;
	eErrorID		:= fbReadHoldingRegistersFc03.eErrorID;
	eExeptionCode	:= fbReadHoldingRegistersFc03.eException;
END_IF;
(* Read Input Registers Fc04 Error *)
IF fbReadInputRegistersFc04.xError AND NOT xErrorHappen THEN
	xErrorHappen 	:= fbReadInputRegistersFc04.xError;
	eErrorID		:= fbReadInputRegistersFc04.eErrorID;
	eExeptionCode	:= fbReadInputRegistersFc04.eException;
END_IF;
(* Write Single Coil Fc05 Error *)
IF fbWriteSingleCoilFc05.xError AND NOT xErrorHappen THEN
	xErrorHappen 	:= fbWriteSingleCoilFc05.xError;
	eErrorID		:= fbWriteSingleCoilFc05.eErrorID;
	eExeptionCode	:= fbWriteSingleCoilFc05.eException;
END_IF;
(* Write Single Register Fc06 Error *)
IF fbWriteSingleRegisterFc06.xError AND NOT xErrorHappen THEN
	xErrorHappen 	:= fbWriteSingleRegisterFc06.xError;
	eErrorID		:= fbWriteSingleRegisterFc06.eErrorID;
	eExeptionCode	:= fbWriteSingleRegisterFc06.eException;
END_IF;		
(* Write Multiple Coils Fc15 Error *)
IF fbWriteMultipleCoilsFc15.xError AND NOT xErrorHappen THEN
	xErrorHappen 	:= fbWriteMultipleCoilsFc15.xError;
	eErrorID		:= fbWriteMultipleCoilsFc15.eErrorID;
	eExeptionCode	:= fbWriteMultipleCoilsFc15.eException;
END_IF;
(* Write Multiple Registers Fc16 Error *)
IF fbWriteMultipleRegistersFc16.xError AND NOT xErrorHappen THEN
	xErrorHappen 	:= fbWriteMultipleRegistersFc16.xError;
	eErrorID		:= fbWriteMultipleRegistersFc16.eErrorID;
	eExeptionCode	:= fbWriteMultipleRegistersFc16.eException;
END_IF;
END_ACTION

PROPERTY P_fbenRTSControl : CtaSysConfig.ITF_BYTE
GET
P_fbenRTSControl := scParameter.fbenRTSControl;
END_GET
END_PROPERTY

ACTION actCallFunctions:
(* Call *)
fbReadCoilsFc01(				rClient := client);				
fbReadDiscreteInputsFc02(		rClient := Client);  
fbReadHoldingRegistersFc03(		rClient := Client);
fbReadInputRegistersFc04(		rClient := Client);	  
fbWriteSingleCoilFc05(			rClient := Client);	  
fbWriteSingleRegisterFc06(		rClient := Client);  
fbWriteMultipleCoilsFc15(		rClient := Client);  
fbWriteMultipleRegistersFc16(	rClient := Client);
END_ACTION

ACTION actCheckBusy:
(* Reset after Busy *)
fbReadCoilsFc01.xExecute				:= fbReadCoilsFc01.xBusy				;
fbReadDiscreteInputsFc02.xExecute	    := fbReadDiscreteInputsFc02.xBusy		;
fbReadHoldingRegistersFc03.xExecute     := fbReadHoldingRegistersFc03.xBusy		;
fbReadInputRegistersFc04.xExecute	    := fbReadInputRegistersFc04.xBusy		;
fbWriteSingleCoilFc05.xExecute		    := fbWriteSingleCoilFc05.xBusy			;
fbWriteSingleRegisterFc06.xExecute	    := fbWriteSingleRegisterFc06.xBusy		;
fbWriteMultipleCoilsFc15.xExecute	    := fbWriteMultipleCoilsFc15.xBusy		;
fbWriteMultipleRegistersFc16.xExecute   := fbWriteMultipleRegistersFc16.xBusy	;
END_ACTION

ACTION actDelays:
(* Delay Read *)
IF _byMbFunction <= 04 THEN
	tonDelay(IN := xTrig,PT := tReadDelay);
(* Delay Write Single *)
ELSIF _byMbFunction >= 5 AND _byMbFunction <= 6 THEN
	tonDelay(IN := xTrig,PT := tWriteDelay); 
(* Delay Write Multiple *)
ELSIF _byMbFunction >= 15 AND _byMbFunction <= 16 THEN
	tonDelay(IN := xTrig,PT := tWriteDelay); 
ELSE 
	tonDelay(IN := xTrig,PT := T#0MS);
END_IF;
END_ACTION

ACTION actExecuteFunction:
(* Read Coils *)
IF _byMbFunction = 01 THEN
	fbReadCoilsFc01.udiReplyTimeout					:= TO_UDINT(tTimeOut) * 1000; 
	fbReadCoilsFc01.udiTimeOut						:= 5000000;
	fbReadCoilsFc01.uiUnitId						:= usiNodeId;
	fbReadCoilsFc01.uiStartItem 					:= TO_UINT(_wMbAdress);
	fbReadCoilsFc01.pData 							:= _pByte;
	fbReadCoilsFc01.uiQuantity						:= TO_UINT(_wQuantity);
	fbReadCoilsFc01.xExecute						:= tonDelay.Q;
(* Read Discret Inputs *)                       	
ELSIF _byMbFunction = 02 THEN                   	
	fbReadDiscreteInputsFc02.udiReplyTimeout		:= TO_UDINT(tTimeOut) * 1000; 
	fbReadDiscreteInputsFc02.udiTimeOut				:= 5000000;
	fbReadDiscreteInputsFc02.uiUnitId				:= usiNodeId;
	fbReadDiscreteInputsFc02.uiStartItem			:= TO_UINT(_wMbAdress);
	fbReadDiscreteInputsFc02.pData 					:= _pByte;
	fbReadDiscreteInputsFc02.uiQuantity				:= TO_UINT(_wQuantity);
	fbReadDiscreteInputsFc02.xExecute				:= tonDelay.Q;
(* Read Holding Registers *)                		
ELSIF _byMbFunction = 03 THEN                   	
	fbReadHoldingRegistersFc03.udiReplyTimeout		:= TO_UDINT(tTimeOut) * 1000; 
	fbReadHoldingRegistersFc03.udiTimeOut			:= 5000000;
	fbReadHoldingRegistersFc03.uiUnitId				:= usiNodeId;          	
	fbReadHoldingRegistersFc03.uiStartItem			:= TO_UINT(_wMbAdress);
	fbReadHoldingRegistersFc03.pData 				:= _pByte;
	fbReadHoldingRegistersFc03.uiQuantity			:= TO_UINT(_wQuantity);
	fbReadHoldingRegistersFc03.xExecute				:= tonDelay.Q;			
(* Read Input Registers *)	                		
ELSIF _byMbFunction = 04 THEN                   	
	fbReadInputRegistersFc04.udiReplyTimeout		:= TO_UDINT(tTimeOut) * 1000; 
	fbReadInputRegistersFc04.udiTimeOut				:= 5000000;
	fbReadInputRegistersFc04.uiUnitId				:= usiNodeId;               	
	fbReadInputRegistersFc04.uiStartItem 			:= TO_UINT(_wMbAdress);
	fbReadInputRegistersFc04.pData 					:= _pByte;
	fbReadInputRegistersFc04.uiQuantity				:= TO_UINT(_wQuantity);
	fbReadInputRegistersFc04.xExecute				:= tonDelay.Q;			
(* Write Single Coil *)	                    		
ELSIF _byMbFunction = 05 THEN                   	
	fbWriteSingleCoilFc05.udiReplyTimeout			:= TO_UDINT(tTimeOut) * 1000; 
	fbWriteSingleCoilFc05.udiTimeOut				:= 5000000;
	fbWriteSingleCoilFc05.uiUnitId					:= usiNodeId;            	
	fbWriteSingleCoilFc05.uiItem 					:= TO_UINT(_wMbAdress);
	fbWriteSingleCoilFc05.xValue 					:= FcBytePointToBoolValue(_pByte);
	fbWriteSingleCoilFc05.xExecute					:= tonDelay.Q;		
(* Write Single Register *)                 		
ELSIF _byMbFunction = 06 THEN                   	
	fbWriteSingleRegisterFc06.udiReplyTimeout		:= TO_UDINT(tTimeOut) * 1000;    
	fbWriteSingleRegisterFc06.udiTimeOut			:= 5000000; 
	fbWriteSingleRegisterFc06.uiUnitId				:= usiNodeId;           	
	fbWriteSingleRegisterFc06.uiItem	  			:= TO_UINT(_wMbAdress);
	fbWriteSingleRegisterFc06.uiValue 				:= FcBytePointToWordValue(_pByte);
	fbWriteSingleRegisterFc06.xExecute				:= tonDelay.Q;		
(* Write Multiple Coils *)		            		
ELSIF _byMbFunction = 15 THEN                   	
	fbWriteMultipleCoilsFc15.udiReplyTimeout		:= TO_UDINT(tTimeOut) * 1000;
	fbWriteMultipleCoilsFc15.udiTimeOut				:= 10000000;
	fbWriteMultipleCoilsFc15.uiUnitId				:= usiNodeId;              	
	fbWriteMultipleCoilsFc15.uiStartItem 			:= TO_UINT(_wMbAdress);
	fbWriteMultipleCoilsFc15.pData 					:= _pByte;
	fbWriteMultipleCoilsFc15.uiQuantity				:= TO_UINT(_wQuantity);
	fbWriteMultipleCoilsFc15.xExecute				:= tonDelay.Q;
(* Write Multiple Registers *)                  	
ELSIF _byMbFunction = 16 THEN                   	
	fbWriteMultipleRegistersFc16.udiReplyTimeout	:= TO_UDINT(tTimeOut) * 1000; 
	fbWriteMultipleRegistersFc16.udiTimeOut			:= 10000000;
	fbWriteMultipleRegistersFc16.uiUnitId			:= usiNodeId;    
	fbWriteMultipleRegistersFc16.uiStartItem 		:= TO_UINT(_wMbAdress);
	fbWriteMultipleRegistersFc16.pData 				:= _pByte;
	fbWriteMultipleRegistersFc16.uiQuantity			:= TO_UINT(_wQuantity);
	fbWriteMultipleRegistersFc16.xExecute			:= tonDelay.Q;	
END_IF;
END_ACTION

PROPERTY P_fbenStopBits : CtaSysConfig.ITF_BYTE
GET
P_fbenStopBits := scParameter.fbenStopBits;
END_GET
END_PROPERTY

PROPERTY P_fbxRtuAscii : CtaSysConfig.ITF_DATATYPE
GET
P_fbxRtuAscii := scParameter.fbxRtuAscii;
END_GET
END_PROPERTY

PROPERTY P_fbbyDataBits : CtaSysConfig.ITF_DATATYPE
GET
P_fbbyDataBits := scParameter.fbbyDataBits;
END_GET
END_PROPERTY

PROPERTY P_fbdwBaudrate : CtaSysConfig.ITF_DATATYPE
GET
P_fbdwBaudrate := scParameter.fbdwBaudrate;
END_GET
END_PROPERTY

PROPERTY P_fbenDTRControl : CtaSysConfig.ITF_BYTE
GET
P_fbenDTRControl := scParameter.fbenDTRControl;
END_GET
END_PROPERTY

PROPERTY P_fbenParity : CtaSysConfig.ITF_BYTE
GET
P_fbenParity := scParameter.fbenParity;
END_GET
END_PROPERTY

PROPERTY P_fbenPort : CtaSysConfig.ITF_INT
GET
P_fbenPort := scParameter.fbenPort;
END_GET
END_PROPERTY

END_FUNCTION_BLOCK

// 21 Interface/CLIENTMANAGER/RTU/ITF_MB_CLIENTMANAGER_RTU
INTERFACE ITF_MB_CLIENTMANAGER_RTU EXTENDS ITF_MB_CLIENTMANAGER

PROPERTY P_fbenStopBits : CtaSysConfig.ITF_BYTE
GET
END_GET
END_PROPERTY

PROPERTY P_fbenPort : CtaSysConfig.ITF_INT
GET
END_GET
END_PROPERTY

PROPERTY P_fbdwBaudrate : CtaSysConfig.ITF_DATATYPE
GET
END_GET
END_PROPERTY

PROPERTY P_fbbyDataBits : CtaSysConfig.ITF_DATATYPE
GET
END_GET
END_PROPERTY

PROPERTY P_fbenParity : CtaSysConfig.ITF_BYTE
GET
END_GET
END_PROPERTY

PROPERTY P_fbenDTRControl : CtaSysConfig.ITF_BYTE
GET
END_GET
END_PROPERTY

PROPERTY P_fbenRTSControl : CtaSysConfig.ITF_BYTE
GET
END_GET
END_PROPERTY

PROPERTY P_fbxRtuAscii : CtaSysConfig.ITF_DATATYPE
GET
END_GET
END_PROPERTY

END_INTERFACE

// 30 Program Organization Units/CLIENT/RTU/FB_MB_CLIENT_RTU
FUNCTION_BLOCK FB_MB_CLIENT_RTU EXTENDS FB_MB_CLIENT IMPLEMENTS ITF_MB_CLIENT_RTU
VAR_OUTPUT
END_VAR
VAR
	(* Config *)
	fbConfigFile				:	CtaSysConfig.fbConfigFile;
	scParameter					:	scSerialClientParameter;
END_VAR

(* Config File *)
actConfig();

PROPERTY TIMEOUT : TIME
GET
TIMEOUT := scParameter.fbtTimeOut.proValue;
END_GET
END_PROPERTY

PROPERTY NODE_ID : USINT
GET
NODE_ID := scParameter.fbusiNodeId.proValue;
END_GET
END_PROPERTY

PROPERTY READ_DELAY : TIME
GET
READ_DELAY := scParameter.fbtReadDelay.proValue;
END_GET
END_PROPERTY

PROPERTY WRITE_DELAY : TIME
GET
WRITE_DELAY := scParameter.fbtWriteDelay.proValue;
END_GET
END_PROPERTY

ACTION actConfig:
(* Config File *)
fbConfigFile();

scParameter.fbxEnable		(_usiParaNr := 1,itfConfigFb := fbConfigFile										);		
scParameter.fbusiNodeId		(_usiParaNr := 2,itfConfigFb := fbConfigFile,_MinInit := 0	 , _MaxInit := 247		);		
scParameter.fbtTimeOut		(_usiParaNr := 3,itfConfigFb := fbConfigFile,_MinInit := T#0MS, _MaxInit := T#5M 	);		
scParameter.fbtReadDelay	(_usiParaNr := 4,itfConfigFb := fbConfigFile,_MinInit := T#0MS, _MaxInit := T#5M 	);		
scParameter.fbtWriteDelay	(_usiParaNr := 5,itfConfigFb := fbConfigFile,_MinInit := T#0MS, _MaxInit := T#5M 	);
END_ACTION

PROPERTY ENABLE : BOOL
GET
ENABLE := scParameter.fbxEnable.proValue;
END_GET
END_PROPERTY

PROPERTY P_fbtReadDelay : CtaSysConfig.ITF_DATATYPE
GET
P_fbtReadDelay := scParameter.fbtReadDelay;
END_GET
END_PROPERTY

PROPERTY P_fbtTimeOut : CtaSysConfig.ITF_DATATYPE
GET
P_fbtTimeOut := scParameter.fbtTimeOut;
END_GET
END_PROPERTY

PROPERTY P_fbtWriteDelay : CtaSysConfig.ITF_DATATYPE
GET
P_fbtWriteDelay := scParameter.fbtWriteDelay;
END_GET
END_PROPERTY

PROPERTY P_fbusiNodeId : CtaSysConfig.ITF_DATATYPE
GET
P_fbusiNodeId := scParameter.fbusiNodeId;
END_GET
END_PROPERTY

PROPERTY P_fbxEnable : CtaSysConfig.ITF_DATATYPE
GET
P_fbxEnable := scParameter.fbxEnable;
END_GET
END_PROPERTY

END_FUNCTION_BLOCK

// 30 Program Organization Units/SERVER/fbModBusServer
{warning 'Each Modbus server needs 400000 bytes of dynamic memory'}
FUNCTION_BLOCK fbModBusServer IMPLEMENTS ITF_SERVER
VAR_INPUT
    I_SerialPort                    :   WagoTypesCom.I_WagoSysComBase;
END_VAR
VAR_OUTPUT
    xError                          :   BOOL;
END_VAR
VAR
    (* Memory *)
    ayxCoil                         :   POINTER TO ARRAY[0..16#FFFF] OF BOOL;
    ayxDiscretInput                 :   POINTER TO ARRAY[0..16#FFFF] OF BOOL;  
    aywInputRegister                :   POINTER TO ARRAY[0..16#FFFF] OF WORD;
    aywHoldingRegister              :   POINTER TO ARRAY[0..16#FFFF] OF WORD; 
    xMemoryError                    :   BOOL;
    xMemoryAllocate                 :   BOOL    := TRUE;
    (* Tcp *)
    fbMbServerModelTcp              :   WagoAppPlcModbus.FbMbSlaveDataModel;
    fbMbShowAccesTcp                :   WagoAppPlcModbus.FbShowMbAccessInfo;
    fbMbTcpServer                   :   WagoAppPlcModbus.FbMbServerTcp;
    scKeepAlive                     :   WagoAppPlcModbus.typKeepAlive;
    ltLastAccesTcp                  :   LTIME;
    fbLastAccesTcp                  :   CtaAppTime.fbTimeMeasurement;
    xErrorWatchDogTcp               :   BOOL;
    xErrorTcp                       :   BOOL;
    
    (* Udp *)
    fbMbServerModelUdp              :   WagoAppPlcModbus.FbMbSlaveDataModel;
    fbMbShowAccesUdp                :   WagoAppPlcModbus.FbShowMbAccessInfo;
    fbMbUdpServer                   :   WagoAppPlcModbus.fbMbServerUdp;
    ltLastAccesUdp                  :   LTIME;
    fbLastAccesUdp                  :   CtaAppTime.fbTimeMeasurement;  
    xErrorWatchDogUdp               :   BOOL;  
    xErrorUdp                       :   BOOL;
    
    (* Serial *)
    fbMbServerModelSerial           :   WagoAppPlcModbus.FbMbSlaveDataModel;
    fbMbShowAccesSerial             :   WagoAppPlcModbus.FbShowMbAccessInfo;
    fbMbRtuSerialServer             :   WagoAppPlcModbus.FbMbServerSerial;
    ltLastAccesSerial               :   LTIME;
    fbLastAccesSerial               :   CtaAppTime.fbTimeMeasurement;
    xErrorWatchDogSerial            :   BOOL;    
    xErrorSerial                    :   BOOL;
    
    (* Parameter *)
    fbConfigFile                    :   CtaSysConfig.fbConfigFile;
    scParameter                     :   scModBusServerParameter;
END_VAR

actConfig();
IF xMemoryAllocate AND NOT xMemoryError THEN
    ayxCoil             := __NEW(BOOL,16#10000);
    ayxDiscretInput     := __NEW(BOOL,16#10000);
    aywInputRegister    := __NEW(WORD,16#10000);
    aywHoldingRegister  := __NEW(WORD,16#10000);
    IF ayxCoil <> 0 AND ayxDiscretInput <> 0 AND aywInputRegister <> 0 AND aywHoldingRegister <> 0 THEN
        xMemoryAllocate     := FALSE;     
    ELSE 
        xMemoryError := TRUE;   
    END_IF;
END_IF;
IF  NOT xMemoryAllocate AND NOT xMemoryError THEN
    IF SIZEOF(ayxCoil^) = 65536 AND SIZEOF(ayxDiscretInput^) = 65536 AND SIZEOF(aywInputRegister^) = 131072 AND SIZEOF(aywHoldingRegister^) = 131072 THEN
        IF NOT fbConfigFile.xError THEN
            actModBusServerSerial();
            actModBusServerTcp();
            actModBusServerUdp();
        END_IF;    
        xMemoryError := FALSE;
    ELSE
        xMemoryError := TRUE;    
    END_IF
END_IF;
(* Error *)
xError := fbConfigFile.xError OR xErrorTcp OR xErrorUdp OR xErrorSerial OR xMemoryError;

ACTION actConfig:
(* Config File *)
fbConfigFile();

scParameter.scSerial.fbbyUnitId            (_usiParaNr :=  1, ItfConfigFb := fbConfigFile , _MinInit :=    0     , _MaxInit :=     247 ); 
scParameter.scSerial.fbxEnable             (_usiParaNr :=  2, ItfConfigFb := fbConfigFile                                              );
scParameter.scSerial.fbudiBaudrate         (_usiParaNr :=  3, ItfConfigFb := fbConfigFile , _MinInit := 9600     , _MaxInit :=   19600 );
scParameter.scSerial.fbusiDataBits         (_usiParaNr :=  4, ItfConfigFb := fbConfigFile , _MinInit :=    5     , _MaxInit :=       8 );
scParameter.scSerial.fbiParity             (_usiParaNr :=  5, ItfConfigFb := fbConfigFile , _MinInit :=    0     , _MaxInit :=       5 );
scParameter.scSerial.fbiStopBits           (_usiParaNr :=  6, ItfConfigFb := fbConfigFile , _MinInit :=    0     , _MaxInit :=       5 );
scParameter.scSerial.fbiHandshake          (_usiParaNr :=  7, ItfConfigFb := fbConfigFile , _MinInit :=    0     , _MaxInit :=       7 );
scParameter.scSerial.fbiPhysikal           (_usiParaNr :=  8, ItfConfigFb := fbConfigFile , _MinInit :=    0     , _MaxInit :=       6 );
scParameter.scSerial.fbxRtuOrAscii         (_usiParaNr :=  9, ItfConfigFb := fbConfigFile                                              );
scParameter.scSerial.fbxEnableWatchDog     (_usiParaNr := 10, ItfConfigFb := fbConfigFile                                              );
scParameter.scSerial.fbtWatchDog           (_usiParaNr := 11, ItfConfigFb := fbConfigFile , _MinInit := T#1S     , _MaxInit :=   T#10M );
scParameter.scTcp.fbxEnable                (_usiParaNr := 12, ItfConfigFb := fbConfigFile                                              );
scParameter.scTcp.fbbyUnitId               (_usiParaNr := 13, ItfConfigFb := fbConfigFile , _MinInit :=    0     , _MaxInit :=     255 ); 
scParameter.scTcp.fbwPort                  (_usiParaNr := 14, ItfConfigFb := fbConfigFile , _MinInit :=    0     , _MaxInit := 16#FFFF );
scParameter.scTcp.fbxKeepAlive             (_usiParaNr := 15, ItfConfigFb := fbConfigFile                                              );
scParameter.scTcp.fbtMaxIdleTime           (_usiParaNr := 16, ItfConfigFb := fbConfigFile , _MinInit := T#1S     , _MaxInit :=   T#10M );
scParameter.scTcp.fbtIntervall             (_usiParaNr := 17, ItfConfigFb := fbConfigFile , _MinInit := T#1S     , _MaxInit :=   T#10M );
scParameter.scTcp.fbudiProbes              (_usiParaNr := 18, ItfConfigFb := fbConfigFile , _MinInit :=    0     , _MaxInit :=     500 );
scParameter.scTcp.fbxEnableWatchDog        (_usiParaNr := 19, ItfConfigFb := fbConfigFile                                              );
scParameter.scTcp.fbtWatchDog              (_usiParaNr := 20, ItfConfigFb := fbConfigFile , _MinInit := T#50MS   , _MaxInit :=   T#10M );
scParameter.scUdp.fbxEnable                (_usiParaNr := 21, ItfConfigFb := fbConfigFile                                              );
scParameter.scUdp.fbbyUnitId               (_usiParaNr := 22, ItfConfigFb := fbConfigFile , _MinInit :=    0     , _MaxInit :=     255 ); 
scParameter.scUdp.fbwPort                  (_usiParaNr := 23, ItfConfigFb := fbConfigFile , _MinInit :=    0     , _MaxInit := 16#FFFF );
scParameter.scUdp.fbxEnableWatchDog        (_usiParaNr := 24, ItfConfigFb := fbConfigFile                                              );
scParameter.scUdp.fbtWatchDog              (_usiParaNr := 25, ItfConfigFb := fbConfigFile , _MinInit := T#1S     , _MaxInit :=   T#10M );
END_ACTION

ACTION actModBusServerTcp:
(* Server Memory Tcp*)
fbMbServerModelTcp(     bUnitId             := scParameter.scTcp.fbbyUnitId.byValue,
                        IIdentifyObject     := GVL_CtaModBus.fbDeviceName,
                        axDiscreteInputs    := ayxDiscretInput^,
                        axCoils             := ayxCoil^,
                        awInputRegisters    := aywInputRegister^,
                        awHoldingRegisters  := aywHoldingRegister^); 
                        
(* Tcp Server *)
IF scParameter.scTcp.fbxEnable.xValue THEN
    scKeepAlive.xEnable                     := scParameter.scTcp.fbxKeepAlive.xValue;
    scKeepAlive.tMaxIdleTime                := scParameter.scTcp.fbtMaxIdleTime.tValue;
    scKeepAlive.tInterval                   := scParameter.scTcp.fbtIntervall.tValue;
    scKeepAlive.udiProbes                   := scParameter.scTcp.fbudiProbes.udiValue;
    fbMbTcpServer(      xOpen               := scParameter.scTcp.fbxEnable.xValue,
                        wPort               := scParameter.scTcp.fbwPort.wValue,
                        utKeepAlive         := scKeepAlive,
                        eFrameType          := WagoAppPlcModbus.eMbFrameType.ETHERNET,
                        I_MbDataModel       := fbMbServerModelTcp.I_MbDataModel);
ELSIF fbMbTcpServer.xOpen THEN
    fbMbTcpServer(      xOpen               := FALSE,
                        I_MbDataModel       := fbMbServerModelTcp.I_MbDataModel);                           
END_IF;                        

(* Acces Info *)
fbMbShowAccesTcp    (   oMbAccessInfo := fbMbServerModelTcp.oMbAccessInfo);   

(* Acces Time *)
IF fbMbServerModelTcp.isReadAccess OR fbMbServerModelTcp.isWriteAccess THEN
    fbLastAccesTcp.Start();
    ltLastAccesTcp := fbLastAccesTcp.Stop();
ELSE
    ltLastAccesTcp := fbLastAccesTcp.Stop();
END_IF;

(* WatchDog *)
IF scParameter.scTcp.fbxEnableWatchDog.xValue THEN
    xErrorWatchDogTcp := TO_LTIME(scParameter.scTcp.fbtWatchDog.tValue) < ltLastAccesTcp;
ELSE
    xErrorWatchDogTcp := FALSE;
END_IF;

(* Error *)
xErrorTcp := fbConfigFile.xError OR fbMbServerModelTcp.xError OR fbMbTcpServer.xError OR xErrorWatchDogTcp;
END_ACTION

ACTION actModBusServerUdp:
(* Server Memory Udp*)
fbMbServerModelUdp(     bUnitId             := scParameter.scUdp.fbbyUnitId.byValue,
                        IIdentifyObject     := GVL_CtaModBus.fbDeviceName,
                        axDiscreteInputs    := ayxDiscretInput^,
                        axCoils             := ayxCoil^,
                        awInputRegisters    := aywInputRegister^,
                        awHoldingRegisters  := aywHoldingRegister^);  
                        
(* UDP Server *)
IF scParameter.scUdp.fbxEnable.xValue THEN
    fbMbUdpServer(      xOpen               := scParameter.scUdp.fbxEnable.xValue,
                        wPort               := scParameter.scUdp.fbwPort.wValue,
                        eFrameType          := WagoAppPlcModbus.eMbFrameType.ETHERNET,
                        I_MbDataModel       := fbMbServerModelUdp.I_MbDataModel);
ELSIF fbMbUdpServer.xOpen THEN
    fbMbUdpServer(      xOpen               := FALSE,
                        I_MbDataModel       := fbMbServerModelUdp.I_MbDataModel);                        
END_IF;                          

(* Acces Info *)
fbMbShowAccesUdp    (   oMbAccessInfo := fbMbServerModelUdp.oMbAccessInfo); 

(* Acces Time *)
IF fbMbServerModelUdp.isReadAccess OR fbMbServerModelUdp.isWriteAccess THEN
    fbLastAccesUdp.Start();
    ltLastAccesUdp := fbLastAccesSerial.Stop();
ELSE
    ltLastAccesUdp := fbLastAccesSerial.Stop();
END_IF;

(* WatchDog *)
IF scParameter.scUdp.fbxEnableWatchDog.xValue THEN
    xErrorWatchDogUdp := TO_LTIME(scParameter.scUdp.fbtWatchDog.tValue) < ltLastAccesUdp;
ELSE
    xErrorWatchDogUdp := FALSE;
END_IF;

(* Error *)
xErrorUdp := fbConfigFile.xError OR fbMbServerModelUdp.xError OR fbMbUdpServer.xError OR xErrorWatchDogUdp;
END_ACTION

ACTION actModBusServerSerial:
(* Server Memory Serial*)
fbMbServerModelSerial(  bUnitId             := scParameter.scSerial.fbbyUnitId.byValue,
                        IIdentifyObject     := GVL_CtaModBus.fbDeviceName,
                        axDiscreteInputs    := ayxDiscretInput^,
                        axCoils             := ayxCoil^,
                        awInputRegisters    := aywInputRegister^,
                        awHoldingRegisters  := aywHoldingRegister^);  
                        
(* SERIAL Server *)           
IF scParameter.scSerial.fbxEnable.xValue THEN    
	IF __QUERYINTERFACE(I_SerialPort,I_SerialPort) THEN
		(* Server Run*) 
		fbMbRtuSerialServer(xConnect            := scParameter.scSerial.fbxEnable.xValue,
							I_Port              := I_SerialPort,
							udiBaudrate         := scParameter.scSerial.fbudiBaudrate.udiValue,
							usiDataBits         := scParameter.scSerial.fbusiDataBits.usiValue,
							eParity             := scParameter.scSerial.fbiParity.iValue,
							eStopBits           := scParameter.scSerial.fbiStopBits.iValue,
							eHandshake          := scParameter.scSerial.fbiHandshake.iValue,
							ePhysical           := scParameter.scSerial.fbiPhysikal.iValue,
							eFrameType          := SEL(scParameter.scSerial.fbxRtuOrAscii.xValue,WagoAppPlcModbus.eMbFrameType.RTU,WagoAppPlcModbus.eMbFrameType.ASCII),
							I_MbDataModel       := fbMbServerModelSerial.I_MbDataModel);
   	END_IF;                     
    (* Acces Info *)
    fbMbShowAccesSerial (   oMbAccessInfo := fbMbServerModelSerial.oMbAccessInfo); 
    
    (* Acces Time *)
    IF fbMbServerModelSerial.isReadAccess OR fbMbServerModelSerial.isWriteAccess THEN
        fbLastAccesSerial.Start();
        ltLastAccesSerial := fbLastAccesSerial.Stop();
    ELSE
        ltLastAccesSerial := fbLastAccesSerial.Stop();
    END_IF;
    
    (* WatchDog *)
    IF scParameter.scSerial.fbxEnableWatchDog.xValue THEN
        xErrorWatchDogSerial := TO_LTIME(scParameter.scSerial.fbtWatchDog.tValue) < ltLastAccesSerial;
    ELSE
        xErrorWatchDogSerial := FALSE;
    END_IF;                        
                        
ELSIF fbMbRtuSerialServer.xConnect THEN
    (* Server Disconnect *)
    fbMbRtuSerialServer(xConnect            := FALSE,
                        I_Port              := I_SerialPort,
                        I_MbDataModel       := fbMbServerModelSerial.I_MbDataModel);   
ELSE
    xErrorWatchDogSerial := FALSE;
    ltLastAccesSerial    := fbLastAccesSerial.Stop();
END_IF;                        



(* Error *)
xErrorSerial := fbConfigFile.xError OR fbMbServerModelSerial.xError OR fbMbRtuSerialServer.xError OR xErrorWatchDogSerial;
END_ACTION

METHOD metGetCoil : BOOL
VAR_INPUT
    wAdr          : WORD;
END_VAR
IF NOT xMemoryAllocate AND NOT xMemoryError THEN
	IF wAdr >= LOWER_BOUND(ayxCoil^,1) AND wAdr <= UPPER_BOUND(ayxCoil^,1) THEN
    	metGetCoil := ayxCoil^[wAdr];
	END_IF;
END_IF;
END_METHOD

METHOD metSetDiscretInput : BOOL
VAR_INPUT
    wAdr          : WORD;
    xValue        : BOOL;
END_VAR
IF NOT xMemoryAllocate AND NOT xMemoryError THEN
	IF wAdr >= LOWER_BOUND(ayxDiscretInput^,1) AND wAdr <= UPPER_BOUND(ayxDiscretInput^,1) THEN
    	ayxDiscretInput^[wAdr] := xValue;
	END_IF;
END_IF;
END_METHOD

METHOD metGetHoldingRegister : WORD
VAR_INPUT
    wAdr          : WORD;
END_VAR
IF NOT xMemoryAllocate AND NOT xMemoryError THEN
	IF wAdr >= LOWER_BOUND(aywHoldingRegister^,1) AND wAdr <= UPPER_BOUND(aywHoldingRegister^,1) THEN
    	metGetHoldingRegister := aywHoldingRegister^[wAdr];
	END_IF;
END_IF;
END_METHOD

METHOD metSetInputRegister : BOOL
VAR_INPUT
    wAdr          : WORD;
    wValue        : WORD;
END_VAR
IF NOT xMemoryAllocate AND NOT xMemoryError THEN
	IF wAdr >= LOWER_BOUND(aywInputRegister^,1) AND wAdr <= UPPER_BOUND(aywInputRegister^,1) THEN
    	aywInputRegister^[wAdr] := wValue;
	END_IF;
END_IF;
END_METHOD

METHOD metAddSerialControll : BOOL
VAR_INPUT
    I_DataAccesListener :   WagoAppPlcModbus.I_DataAccessListener;
END_VAR
fbMbServerModelSerial.RegisterDataAccessListener(I_DataAccesListener);
END_METHOD

METHOD metAddTcpControll : BOOL
VAR_INPUT
    I_DataAccesListener :   WagoAppPlcModbus.I_DataAccessListener;
END_VAR
fbMbServerModelTcp.RegisterDataAccessListener(I_DataAccesListener);
END_METHOD

METHOD metAddUdpControll : BOOL
VAR_INPUT
    I_DataAccesListener :   WagoAppPlcModbus.I_DataAccessListener;
END_VAR
fbMbServerModelUdp.RegisterDataAccessListener(I_DataAccesListener);
END_METHOD

METHOD metSetHoldingRegister : BOOL
VAR_INPUT
    wAdr          : WORD;
    wValue        : WORD;
END_VAR
IF NOT xMemoryAllocate AND NOT xMemoryError THEN
	IF wAdr >= LOWER_BOUND(aywHoldingRegister^,1) AND wAdr <= UPPER_BOUND(aywHoldingRegister^,1) THEN
    	aywHoldingRegister^[wAdr] := wValue;
	END_IF;
END_IF;
END_METHOD

METHOD metSetCoil : BOOL
VAR_INPUT
    wAdr          : WORD;
    xValue        : BOOL;
END_VAR
IF NOT xMemoryAllocate AND NOT xMemoryError THEN
	IF wAdr >= LOWER_BOUND(ayxCoil^,1) AND wAdr <= UPPER_BOUND(ayxCoil^,1) THEN
    	ayxCoil^[wAdr] := xValue;
	END_IF;
END_IF;
END_METHOD

END_FUNCTION_BLOCK

// 21 Interface/SERVER/ITF_SERVER
INTERFACE ITF_SERVER EXTENDS __SYSTEM.IQueryInterface

METHOD metGetCoil : BOOL
VAR_INPUT
    wAdr          : WORD;
END_VAR
END_METHOD

METHOD metGetHoldingRegister : WORD
VAR_INPUT
    wAdr          : WORD;
END_VAR
END_METHOD

METHOD metSetCoil : BOOL
VAR_INPUT
    wAdr          : WORD;
    xValue        : BOOL;
END_VAR
END_METHOD

METHOD metSetDiscretInput : BOOL
VAR_INPUT
    wAdr          : WORD;
    xValue        : BOOL;
END_VAR
END_METHOD

METHOD metSetHoldingRegister : BOOL
VAR_INPUT
    wAdr          : WORD;
    wValue        : WORD;
END_VAR
END_METHOD

METHOD metSetInputRegister : BOOL
VAR_INPUT
    wAdr          : WORD;
    wValue        : WORD;
END_VAR
END_METHOD

END_INTERFACE

// 30 Program Organization Units/SERVER/FB_SERVER
{attribute 'no_assign'}
FUNCTION_BLOCK FB_SERVER IMPLEMENTS ITF_SERVER_PARA
VAR_INPUT
END_VAR
VAR_OUTPUT
END_VAR
VAR
	(* Servers *)	
	fbServerTcp						:	ModbusFB.ServerTCP;
	fbServerSerial					:	ModbusFB.ServerSerial;
	(* Data *)
    ayxCoil                         :   ARRAY[0..16#FFFF] OF BOOL;
    ayxDiscretInput                 :   ARRAY[0..16#FFFF] OF BOOL;  
    aywInputRegister                :   ARRAY[0..16#FFFF] OF WORD;
    aywHoldingRegister              :   ARRAY[0..16#FFFF] OF WORD; 	
	
	(* Data Model *)
	scDataModel						:	ModbusFB.TableDefinitions;
	scSectionCoil					:	ARRAY[0..1] OF ModbusFB.TableSection;
	scSectionDiscretInput			:	ARRAY[0..1] OF ModbusFB.TableSection;
	scSectionInputRegister			:	ARRAY[0..1] OF ModbusFB.TableSection;
	scSectionHoldingRegister		:	ARRAY[0..1] OF ModbusFB.TableSection;
	
	(* Help Variable *)
	xEnableTcp						:	BOOL;
	xEnableSerial					:	BOOL;

	(* Config *)
	fbConfigFile					:	CtaSysConfig.fbConfigFile;
	scParameter						:	scModBusServerParameter;
END_VAR

(* Config *)
actConfig();

(* DataModell *)
actDataModel();

(* TCP Server *)
fbServerTcp(	xEnable	 				:= xEnableTcp,
				dataModel 				:= scDataModel,
				tInactivityInfoTime		:= TO_UDINT(T#1M),
				wsInterfaceName			:= TO_WSTRING(scParameter.scTcp.fbstInterface.proValue),
				uiPort					:= TO_UINT(scParameter.scTcp.fbwPort.proValue),
				xReset					:= fbServerTcp.xError,
				udiLogOptions			:= );
	
(* Serial Server *)
fbServerSerial(	xEnable	 				:= xEnableSerial,
				dataModel 				:= scDataModel,
				tInactivityInfoTime		:= TO_UDINT(T#1M),
				uiUnitId				:= TO_UINT(scParameter.scSerial.fbusiNodeId.proValue),
				iPort					:= scParameter.scSerial.fbenPort.proValue,
				dwBaudrate				:= scParameter.scSerial.fbdwBaudrate.proValue,
				byDataBits				:= scParameter.scSerial.fbbyDataBits.proValue,
				eParity					:= scParameter.scSerial.fbenParity.proValue,
				eStopBits				:= scParameter.scSerial.fbenStopBits.proValue,
				eDTRcontrol				:= scParameter.scSerial.fbenDTRControl.proValue,
				eRTScontrol				:= scParameter.scSerial.fbenRTSControl.proValue,
				eRtuAscii				:= SEL(scParameter.scSerial.fbxRtuAscii.proValue,ModbusFB.RtuAscii.RTU,ModbusFB.RtuAscii.ASCII),
				udiLogOptions			:= );

ACTION actConfig:
(* Config File *)
fbConfigFile();

scParameter.scSerial.fbxEnable              (_usiParaNr :=  1, ItfConfigFb := fbConfigFile                                              );
scParameter.scSerial.fbusiNodeId            (_usiParaNr :=  2, ItfConfigFb := fbConfigFile , _MinInit :=    0     , _MaxInit :=     247 ); 
scParameter.scSerial.fbdwBaudrate           (_usiParaNr :=  3, ItfConfigFb := fbConfigFile , _MinInit := 9600     , _MaxInit :=   19600 );
scParameter.scSerial.fbbyDataBits           (_usiParaNr :=  4, ItfConfigFb := fbConfigFile , _MinInit :=    5     , _MaxInit :=       8 );
scParameter.scSerial.fbenParity             (_usiParaNr :=  5, ItfConfigFb := fbConfigFile , _MinInit :=    0     , _MaxInit :=       5 );
scParameter.scSerial.fbenStopBits           (_usiParaNr :=  6, ItfConfigFb := fbConfigFile , _MinInit :=    0     , _MaxInit :=       5 );
scParameter.scSerial.fbenDTRControl         (_usiParaNr :=  7, ItfConfigFb := fbConfigFile , _MinInit :=    0     , _MaxInit :=       2 );
scParameter.scSerial.fbenRTSControl         (_usiParaNr :=  8, ItfConfigFb := fbConfigFile , _MinInit :=    0     , _MaxInit :=       2 );
scParameter.scSerial.fbxRtuAscii            (_usiParaNr :=  9, ItfConfigFb := fbConfigFile                                              );
scParameter.scSerial.fbxEnableWatchDog      (_usiParaNr := 10, ItfConfigFb := fbConfigFile                                              );
scParameter.scSerial.fbtWatchDog            (_usiParaNr := 11, ItfConfigFb := fbConfigFile , _MinInit := T#1S     , _MaxInit :=   T#10M );
scParameter.scTcp.fbxEnable                 (_usiParaNr := 12, ItfConfigFb := fbConfigFile                                              );
scParameter.scTcp.fbwPort                   (_usiParaNr := 13, ItfConfigFb := fbConfigFile , _MinInit :=    0     , _MaxInit := 16#FFFF );
scParameter.scTcp.fbxEnableWatchDog         (_usiParaNr := 14, ItfConfigFb := fbConfigFile                                              );
scParameter.scTcp.fbtWatchDog               (_usiParaNr := 15, ItfConfigFb := fbConfigFile , _MinInit := T#50MS   , _MaxInit :=   T#10M );
scParameter.scTcp.fbstInterface				(_usiParaNr := 16, ItfConfigFb := fbConfigFile 												);





(* Serial Change reset enable*)
IF scParameter.scSerial.fbxEnable.proStateChanged         	OR
   scParameter.scSerial.fbusiNodeId.proStateChanged       	OR
   scParameter.scSerial.fbdwBaudrate.proStateChanged      	OR 
   scParameter.scSerial.fbbyDataBits.proStateChanged      	OR 
   scParameter.scSerial.fbenParity.proStateChanged       	OR 
   scParameter.scSerial.fbenStopBits.proStateChanged     	OR 
   scParameter.scSerial.fbenDTRControl.proStateChanged    	OR 
   scParameter.scSerial.fbenRTSControl.proStateChanged    	OR 
   scParameter.scSerial.fbxRtuAscii.proStateChanged      	OR 
   scParameter.scSerial.fbxEnableWatchDog.proStateChanged 	OR 
   scParameter.scSerial.fbtWatchDog.proStateChanged       	THEN
	xEnableSerial := FALSE;
ELSE
	xEnableSerial := scParameter.scSerial.fbxEnable.proValue;
END_IF;

(* Tcp Change reset enable*)
IF scParameter.scTcp.fbxEnable.proStateChanged				OR     
   scParameter.scTcp.fbwPort.proStateChanged				OR                                
   scParameter.scTcp.fbxEnableWatchDog.proStateChanged		OR  
   scParameter.scTcp.fbtWatchDog.proStateChanged			OR  
   scParameter.scTcp.fbstInterface.proStateChanged			THEN	
	xEnableTcp := FALSE;
ELSE
	xEnableTcp := scParameter.scTcp.fbxEnable.proValue;
END_IF;
END_ACTION

METHOD metGetCoil : BOOL
VAR_INPUT
	wAdr	: WORD;
END_VAR
IF wAdr >= 0 AND wAdr <= 16#FFFF THEN
	metGetCoil := ayxCoil[wAdr];
END_IF;
END_METHOD

METHOD metGetHoldingRegister : WORD
VAR_INPUT
	wAdr	: WORD;
END_VAR
IF wAdr >= 0 AND wAdr <= 16#FFFF THEN
	metGetHoldingRegister := aywHoldingRegister[wAdr];
END_IF;
END_METHOD

METHOD metSetCoil : BOOL
VAR_INPUT
	wAdr	: WORD;
	xValue	: BOOL;
END_VAR
IF wAdr >= 0 AND wAdr <= 16#FFFF THEN
	ayxCoil[wAdr] := xValue ;
	metSetCoil := TRUE;
END_IF;
END_METHOD

METHOD metSetDiscretInput : BOOL
VAR_INPUT
	wAdr	: WORD;
	xValue	: BOOL;
END_VAR
IF wAdr >= 0 AND wAdr <= 16#FFFF THEN
	ayxDiscretInput[wAdr] := xValue ;
	metSetDiscretInput := TRUE;
END_IF;
END_METHOD

METHOD metSetHoldingRegister : BOOL
VAR_INPUT
	wAdr	: WORD;
	wValue	: WORD;
END_VAR
IF wAdr >= 0 AND wAdr <= 16#FFFF THEN
	aywHoldingRegister[wAdr] := wValue ;
	metSetHoldingRegister := TRUE;
END_IF;
END_METHOD

METHOD metSetInputRegister : BOOL
VAR_INPUT
	wAdr	: WORD;
	wValue	: WORD;
END_VAR
IF wAdr >= 0 AND wAdr <= 16#FFFF THEN
	aywInputRegister[wAdr] := wValue ;
	metSetInputRegister := TRUE;
END_IF;
END_METHOD

ACTION actDataModel:
(* Coil Data Model *)
scSectionCoil[0].pStartAddr						:= ADR(ayxCoil[0]);
scSectionCoil[0].uiStart						:= 0;
scSectionCoil[0].uiNumDataItems					:= 16#0001;
scSectionCoil[0].uiDataItemSize					:= 1;
scSectionCoil[1].pStartAddr						:= ADR(ayxCoil[1]);
scSectionCoil[1].uiStart						:= 1;
scSectionCoil[1].uiNumDataItems					:= 16#FFFF;
scSectionCoil[1].uiDataItemSize					:= 1;

scDataModel.tableCoils.pSections 				:= ADR(scSectionCoil);
scDataModel.tableCoils.uiNumSections			:= 2;

(* Discret Input Data Model *)
scSectionDiscretInput[0].pStartAddr				:= ADR(ayxDiscretInput[0]);
scSectionDiscretInput[0].uiStart				:= 0;
scSectionDiscretInput[0].uiNumDataItems			:= 16#0001;
scSectionDiscretInput[0].uiDataItemSize			:= 1;
scSectionDiscretInput[1].pStartAddr				:= ADR(ayxDiscretInput[1]);
scSectionDiscretInput[1].uiStart				:= 1;
scSectionDiscretInput[1].uiNumDataItems			:= 16#FFFF;
scSectionDiscretInput[1].uiDataItemSize			:= 1;

scDataModel.tableDiscreteInputs.pSections		:= ADR(scSectionDiscretInput);
scDataModel.tableDiscreteInputs.uiNumSections	:= 2;

(* Holding Register Data Model *)
scSectionHoldingRegister[0].pStartAddr			:= ADR(aywHoldingRegister[0]);
scSectionHoldingRegister[0].uiStart				:= 0;
scSectionHoldingRegister[0].uiNumDataItems		:= 16#0001;
scSectionHoldingRegister[0].uiDataItemSize		:= 16;
scSectionHoldingRegister[1].pStartAddr			:= ADR(aywHoldingRegister[1]);
scSectionHoldingRegister[1].uiStart				:= 1;
scSectionHoldingRegister[1].uiNumDataItems		:= 16#FFFF;
scSectionHoldingRegister[1].uiDataItemSize		:= 16;

scDataModel.tableHoldingRegisters.pSections		:= ADR(scSectionHoldingRegister);
scDataModel.tableHoldingRegisters.uiNumSections := 2;

(* Input Register Data Model *)
scSectionInputRegister[0].pStartAddr			:= ADR(aywInputRegister[0]);
scSectionInputRegister[0].uiStart				:= 0;
scSectionInputRegister[0].uiNumDataItems		:= 16#0001;
scSectionInputRegister[0].uiDataItemSize		:= 16;
scSectionInputRegister[1].pStartAddr			:= ADR(aywInputRegister[1]);
scSectionInputRegister[1].uiStart				:= 1;
scSectionInputRegister[1].uiNumDataItems		:= 16#FFFF;
scSectionInputRegister[1].uiDataItemSize		:= 16;

scDataModel.tableInputRegisters.pSections		:= ADR(scSectionInputRegister);
scDataModel.tableInputRegisters.uiNumSections	:= 2;
END_ACTION

PROPERTY P_Serial_fbbyDataBits : CtaSysConfig.ITF_BYTE
GET
P_Serial_fbbyDataBits := scParameter.scSerial.fbbyDataBits;
END_GET
END_PROPERTY

PROPERTY P_Serial_fbdwBaudrate : CtaSysConfig.ITF_DWORD
GET
P_Serial_fbdwBaudrate := scParameter.scSerial.fbdwBaudrate;
END_GET
END_PROPERTY

